// TwinCAT 3 PLC project AstroBROTTests
// Title: AstroBROTTests
// Company: BROT
// ProjectVersion: 0.1.0
// ProgramVersion: 3.1.4024.66
// libraries:
//   AstroBROT, * (BROT)
//   Tc2_Standard, * (Beckhoff Automation GmbH)
//   Tc2_System, * (Beckhoff Automation GmbH)
//   Tc2_Utilities, * (Beckhoff Automation GmbH)
//   Tc3_Module, * (Beckhoff Automation GmbH)
//   TcUnit, * (www.tcunit.org)
// project tree:
//   / PlcTask.TcTTO (not stored)
//   POUs/ FB_DateTime2JD_Tests.TcPOU, FB_ATAN2_Tests.TcPOU, FB_ALTAZ2HADEC_Tests.TcPOU, FB_CO_ABERRATION_Tests.TcPOU, FB_CO_NUTATE_Tests.TcPOU, FB_CO_REFRACT_Tests.TcPOU, FB_DUT1_Tests.TcPOU, FB_Pipeline_Tests.TcPOU, FB_JD2LST_Tests.TcPOU, FB_EQ2HOR_Tests.TcPOU, FB_HOR2EQ_Tests.TcPOU, FB_TEN_Tests.TcPOU, FB_PRECESS_Tests.TcPOU, FB_RADEC2HADEC_Tests.TcPOU, FB_HADEC2RADEC_Tests.TcPOU, FB_SUNPOS_Tests.TcPOU, FB_EdgeCases_Tests.TcPOU, MAIN.TcPOU
// real-time tasks:
//   TASK PlcTask: cycle T#10ms, priority 20, ADS port 350

// ---- POUs/FB_DateTime2JD_Tests.TcPOU
// Tests for AstroBROT.DateTime2JD (TIMESTRUCT, UTC, to Julian Date).
//
// Golden values come from erfa.cal2jd (Gregorian calendar), tolerance 1e-8 days (0.9 ms).
FUNCTION_BLOCK FB_DateTime2JD_Tests EXTENDS TcUnit.FB_TestSuite
VAR
END_VAR

Golden_Dates();
Leap_Years();
Milliseconds();
Out_Of_Range_Fields_Roll_Over();

METHOD PRIVATE Jd : LREAL
VAR_INPUT
	wYear, wMonth, wDay, wHour, wMinute, wSecond, wMilliseconds	: UINT;
END_VAR
VAR
	t	: TIMESTRUCT;
END_VAR
t.wYear := wYear;
t.wMonth := wMonth;
t.wDay := wDay;
t.wHour := wHour;
t.wMinute := wMinute;
t.wSecond := wSecond;
t.wMilliseconds := wMilliseconds;
Jd := AstroBROT.DateTime2JD(epoch := t);
END_METHOD

METHOD PRIVATE CheckNear
VAR_INPUT
	fExpected	: LREAL;
	fActual		: LREAL;
	fDelta		: LREAL;
	sName		: STRING(255);
END_VAR
AssertEquals_LREAL(Expected := fExpected, Actual := fActual, Delta := fDelta, Message := sName);
END_METHOD

METHOD PRIVATE Golden_Dates
VAR
END_VAR
TEST('Golden_Dates');
CheckNear(2451545.0, Jd(2000, 1, 1, 12, 0, 0, 0), 1.0E-8, 'J2000');
CheckNear(2461304.5, Jd(2026, 9, 21, 0, 0, 0, 0), 1.0E-8, '2026-09-21 00:00');
CheckNear(2461305.2710069446, Jd(2026, 9, 21, 18, 30, 15, 0), 1.0E-8, '2026-09-21 18:30:15');
CheckNear(2451544.499988426, Jd(1999, 12, 31, 23, 59, 59, 0), 1.0E-8, '1999-12-31 23:59:59');
CheckNear(2299160.5, Jd(1582, 10, 15, 0, 0, 0, 0), 1.0E-8, '1582-10-15, first Gregorian day');
TEST_FINISHED();
END_METHOD

METHOD PRIVATE Leap_Years
VAR
END_VAR
TEST('Leap_Years');
CheckNear(2460370.0, Jd(2024, 2, 29, 12, 0, 0, 0), 1.0E-8, '2024-02-29 12:00');
CheckNear(1.0, Jd(2024, 3, 1, 0, 0, 0, 0) - Jd(2024, 2, 29, 0, 0, 0, 0), 1.0E-9, '2024 is a leap year');
CheckNear(1.0, Jd(2100, 3, 1, 0, 0, 0, 0) - Jd(2100, 2, 28, 0, 0, 0, 0), 1.0E-9, '2100 is not a leap year');
CheckNear(1.0, Jd(2000, 3, 1, 0, 0, 0, 0) - Jd(2000, 2, 29, 0, 0, 0, 0), 1.0E-9, '2000 is a leap year');
TEST_FINISHED();
END_METHOD

METHOD PRIVATE Milliseconds
VAR
END_VAR
TEST('Milliseconds');
// 500 ms = 5.787037037037037E-6 days
CheckNear(5.787037037037037E-6, Jd(2026, 9, 21, 0, 0, 0, 500) - Jd(2026, 9, 21, 0, 0, 0, 0), 1.0E-9, '500 ms');
CheckNear(1.1574074074074073E-8, Jd(2026, 9, 21, 0, 0, 0, 1) - Jd(2026, 9, 21, 0, 0, 0, 0), 1.0E-9, '1 ms');
TEST_FINISHED();
END_METHOD

METHOD PRIVATE Out_Of_Range_Fields_Roll_Over
VAR
END_VAR
TEST('Out_Of_Range_Fields_Roll_Over');
// documented behaviour, not a feature to rely on
CheckNear(2461406.5, Jd(2026, 13, 1, 0, 0, 0, 0), 1.0E-8, 'month 13 is January of the next year');
CheckNear(2461101.5, Jd(2026, 2, 30, 0, 0, 0, 0), 1.0E-8, '30 February is 2 March');
TEST_FINISHED();
END_METHOD

END_FUNCTION_BLOCK

// ---- POUs/FB_ATAN2_Tests.TcPOU
// Tests for AstroBROT.ATAN2, the four-quadrant arctangent (TwinCAT's PLC has none of its own).
//
// Expected values come from Python math.atan2, tolerance 1e-12 rad. Known difference from IEEE: y = -0.0 with x < 0
// gives +pi (ST cannot tell -0.0 from 0.0), harmless because the callers wrap the angle.
FUNCTION_BLOCK FB_ATAN2_Tests EXTENDS TcUnit.FB_TestSuite
VAR
END_VAR

Quadrants();
Axes();
Origin_Is_Zero();
Close_To_The_Axes();

METHOD PRIVATE CheckAtan2
VAR_INPUT
	fExpected	: LREAL;
	fActual		: LREAL;
	sName		: STRING(255);
END_VAR
AssertEquals_LREAL(Expected := fExpected, Actual := fActual, Delta := 1.0E-12, Message := sName);
END_METHOD

METHOD PRIVATE Quadrants
VAR
END_VAR
TEST('Quadrants');
CheckAtan2(0.7853981633974483, AstroBROT.ATAN2(y := 1.0, x := 1.0), 'q1 (1, 1)');
CheckAtan2(2.5535900500422257, AstroBROT.ATAN2(y := 2.0, x := -3.0), 'q2 (2, -3)');
CheckAtan2(-2.5535900500422257, AstroBROT.ATAN2(y := -2.0, x := -3.0), 'q3 (-2, -3)');
CheckAtan2(-0.5880026035475675, AstroBROT.ATAN2(y := -2.0, x := 3.0), 'q4 (-2, 3)');
CheckAtan2(0.5880026035475675, AstroBROT.ATAN2(y := 2.0, x := 3.0), 'q1 (2, 3)');
CheckAtan2(2.356194490192345, AstroBROT.ATAN2(y := 1.0, x := -1.0), 'q2 (1, -1)');
CheckAtan2(-2.356194490192345, AstroBROT.ATAN2(y := -1.0, x := -1.0), 'q3 (-1, -1)');
CheckAtan2(-0.7853981633974483, AstroBROT.ATAN2(y := -1.0, x := 1.0), 'q4 (-1, 1)');
TEST_FINISHED();
END_METHOD

METHOD PRIVATE Axes
VAR
END_VAR
TEST('Axes');
CheckAtan2(0.0, AstroBROT.ATAN2(y := 0.0, x := 1.0), '+x axis');
CheckAtan2(1.5707963267948966, AstroBROT.ATAN2(y := 1.0, x := 0.0), '+y axis');
CheckAtan2(-1.5707963267948966, AstroBROT.ATAN2(y := -1.0, x := 0.0), '-y axis');
CheckAtan2(3.141592653589793, AstroBROT.ATAN2(y := 0.0, x := -1.0), '-x axis, y = 0 gives +pi');
TEST_FINISHED();
END_METHOD

METHOD PRIVATE Origin_Is_Zero
VAR
END_VAR
TEST('Origin_Is_Zero');
CheckAtan2(0.0, AstroBROT.ATAN2(y := 0.0, x := 0.0), 'origin');
TEST_FINISHED();
END_METHOD

METHOD PRIVATE Close_To_The_Axes
VAR
END_VAR
TEST('Close_To_The_Axes');
CheckAtan2(1.5707963267938967, AstroBROT.ATAN2(y := 1.0, x := 1.0E-12), 'just right of the +y axis');
CheckAtan2(3.141592653588793, AstroBROT.ATAN2(y := 1.0E-12, x := -1.0), 'just above the -x axis');
CheckAtan2(-3.141592653588793, AstroBROT.ATAN2(y := -1.0E-12, x := -1.0), 'just below the -x axis');
TEST_FINISHED();
END_METHOD

END_FUNCTION_BLOCK

// ---- POUs/FB_ALTAZ2HADEC_Tests.TcPOU
// Tests for AstroBROT.FB_ALTAZ2HADEC.
//
// At the celestial pole (az = 0, alt = lat; or az = 180, alt = -lat for the south pole) the argument of ASIN is
// exactly 1 in theory, but rounding gives 1 + 2.2E-16 for many latitudes, and ASIN of that is NaN (issue #18).
FUNCTION_BLOCK FB_ALTAZ2HADEC_Tests EXTENDS TcUnit.FB_TestSuite
VAR
END_VAR

Ordinary_Position();
Pointing_At_The_North_Pole();
Pointing_At_The_South_Pole();

METHOD PRIVATE Ordinary_Position
VAR
	fb	: AstroBROT.FB_ALTAZ2HADEC;
END_VAR
TEST('Ordinary_Position');
// sin(dec) = sin(45)^2 + 0 = 0.5, so dec = 30 deg
fb(alt := 45.0, az := 90.0, lat := 45.0);
AssertEquals_LREAL(Expected := 30.0, Actual := fb.dec, Delta := 1.0E-9, Message := 'dec at alt 45, az 90, lat 45');
TEST_FINISHED();
END_METHOD

METHOD PRIVATE Pointing_At_The_North_Pole
VAR
	fb	: AstroBROT.FB_ALTAZ2HADEC;
END_VAR
TEST('Pointing_At_The_North_Pole');
fb(alt := 45.0, az := 0.0, lat := 45.0);
AssertTrue(Condition := ABS(fb.dec - 90.0) < 1.0E-6, Message := 'lat 45 north pole, dec is 90 (and not NaN)');
fb(alt := 34.0, az := 0.0, lat := 34.0);
AssertTrue(Condition := ABS(fb.dec - 90.0) < 1.0E-6, Message := 'lat 34 north pole, dec is 90 (and not NaN)');
fb(alt := 58.0, az := 0.0, lat := 58.0);
AssertTrue(Condition := ABS(fb.dec - 90.0) < 1.0E-6, Message := 'lat 58 north pole, dec is 90 (and not NaN)');
fb(alt := -34.0, az := 0.0, lat := -34.0);
AssertTrue(Condition := ABS(fb.dec - 90.0) < 1.0E-6, Message := 'lat -34 north pole, dec is 90 (and not NaN)');
TEST_FINISHED();
END_METHOD

METHOD PRIVATE Pointing_At_The_South_Pole
VAR
	fb	: AstroBROT.FB_ALTAZ2HADEC;
END_VAR
TEST('Pointing_At_The_South_Pole');
fb(alt := -45.0, az := 180.0, lat := 45.0);
AssertTrue(Condition := ABS(fb.dec + 90.0) < 1.0E-6, Message := 'lat 45 south pole, dec is -90 (and not NaN)');
fb(alt := -34.0, az := 180.0, lat := 34.0);
AssertTrue(Condition := ABS(fb.dec + 90.0) < 1.0E-6, Message := 'lat 34 south pole, dec is -90 (and not NaN)');
fb(alt := -58.0, az := 180.0, lat := 58.0);
AssertTrue(Condition := ABS(fb.dec + 90.0) < 1.0E-6, Message := 'lat 58 south pole, dec is -90 (and not NaN)');
fb(alt := 34.0, az := 180.0, lat := -34.0);
AssertTrue(Condition := ABS(fb.dec + 90.0) < 1.0E-6, Message := 'lat -34 south pole, dec is -90 (and not NaN)');
TEST_FINISHED();
END_METHOD

END_FUNCTION_BLOCK

// ---- POUs/FB_CO_ABERRATION_Tests.TcPOU
// Tests for AstroBROT.FB_CO_ABERRATION (annual aberration, Meeus chapter 23).
//
// ra/dec are the coordinates precessed to the date, eps = 0 means "calculate the obliquity from jd". Golden values
// come from AstroBROT/testing/golden_astro.py. Tolerance 1e-9 deg (3.6 uas).
FUNCTION_BLOCK FB_CO_ABERRATION_Tests EXTENDS TcUnit.FB_TestSuite
VAR
END_VAR

Golden_Tenerife_2026();
Golden_South_2010();
Eps_Input_Is_Not_Modified();

METHOD PRIVATE CheckNear
VAR_INPUT
	fExpected	: LREAL;
	fActual		: LREAL;
	fDelta		: LREAL;
	sName		: STRING(255);
END_VAR
AssertEquals_LREAL(Expected := fExpected, Actual := fActual, Delta := fDelta, Message := sName);
END_METHOD

METHOD PRIVATE CheckAngle
VAR_INPUT
	fExpected	: LREAL;
	fActual		: LREAL;
	fDelta		: LREAL;
	sName		: STRING(255);
END_VAR
VAR
	fDiff	: LREAL;
END_VAR
// angles in degrees, compared modulo 360 so that 359.9999999 and -1.0E-7 are equal
fDiff := fActual - fExpected;
WHILE fDiff > 180.0 DO fDiff := fDiff - 360.0; END_WHILE
WHILE fDiff < -180.0 DO fDiff := fDiff + 360.0; END_WHILE
AssertEquals_LREAL(Expected := 0.0, Actual := fDiff, Delta := fDelta, Message := sName);
END_METHOD

METHOD PRIVATE Golden_Tenerife_2026
VAR
	fbCalc	: AstroBROT.FB_CO_ABERRATION;
	fbGiven	: AstroBROT.FB_CO_ABERRATION;
END_VAR
TEST('Golden_Tenerife_2026');
fbCalc(jd := 2461300.75, ra := 84.03200262159413, dec := 22.025976570150018, eps := 0.0);
CheckAngle(8.195455011719691e-05, fbCalc.d_ra, 1.0E-9, 'Tenerife_2026 d_ra, eps calculated');
CheckNear(0.00013148215303962214, fbCalc.d_dec, 1.0E-9, 'Tenerife_2026 d_dec, eps calculated');
fbGiven(jd := 2461300.75, ra := 84.03200262159413, dec := 22.025976570150018, eps := 0.40907226011280384);
CheckAngle(8.195455011719691e-05, fbGiven.d_ra, 1.0E-9, 'Tenerife_2026 d_ra, eps given');
CheckNear(0.00013148215303962214, fbGiven.d_dec, 1.0E-9, 'Tenerife_2026 d_dec, eps given');
TEST_FINISHED();
END_METHOD

METHOD PRIVATE Golden_South_2010
VAR
	fbCalc	: AstroBROT.FB_CO_ABERRATION;
	fbGiven	: AstroBROT.FB_CO_ABERRATION;
END_VAR
TEST('Golden_South_2010');
fbCalc(jd := 2455197.5, ra := 312.6725080638107, dec := -47.262327080321406, eps := 0.0);
CheckAngle(-0.007132163801626435, fbCalc.d_ra, 1.0E-9, 'South_2010 d_ra, eps calculated');
CheckNear(-0.0025955563049355266, fbCalc.d_dec, 1.0E-9, 'South_2010 d_dec, eps calculated');
fbGiven(jd := 2455197.5, ra := 312.6725080638107, dec := -47.262327080321406, eps := 0.4090837545317484);
CheckAngle(-0.007132163801626435, fbGiven.d_ra, 1.0E-9, 'South_2010 d_ra, eps given');
CheckNear(-0.0025955563049355266, fbGiven.d_dec, 1.0E-9, 'South_2010 d_dec, eps given');
TEST_FINISHED();
END_METHOD

METHOD PRIVATE Eps_Input_Is_Not_Modified
VAR
	fb	: AstroBROT.FB_CO_ABERRATION;
END_VAR
TEST('Eps_Input_Is_Not_Modified');
// with eps = 0 the block calculates the obliquity itself; it used to store the result in its input, so the
// value of the first jd was reused for every later call
fb(jd := 2461300.75, ra := 84.03200262159413, dec := 22.025976570150018, eps := 0.0);
CheckNear(0.0, fb.eps, 1.0E-15, 'eps stays 0 after the call');
fb(jd := 2455197.5, ra := 312.6725080638107, dec := -47.262327080321406, eps := 0.0);
CheckNear(0.0, fb.eps, 1.0E-15, 'eps stays 0 after the second call');
CheckAngle(-0.007132163801626435, fb.d_ra, 1.0E-9, 'second epoch d_ra');
CheckNear(-0.0025955563049355266, fb.d_dec, 1.0E-9, 'second epoch d_dec');
TEST_FINISHED();
END_METHOD

END_FUNCTION_BLOCK

// ---- POUs/FB_CO_NUTATE_Tests.TcPOU
// Tests for AstroBROT.FB_CO_NUTATE (RA/Dec corrections due to nutation).
//
// Golden values come from AstroBROT/testing/astrobrot_port.py (co_nutate), tolerance 1e-7 deg.
// Issue #10: d_ra was ra2 - ra with ra2 in [0, 360) and ra unwrapped, so ra = -5 gave d_ra = 360.0004 instead of
// 0.00035. The fix wraps d_ra to [-180, 180).
FUNCTION_BLOCK FB_CO_NUTATE_Tests EXTENDS TcUnit.FB_TestSuite
VAR
END_VAR

Golden_Ra_Minus_5();
Golden_Ra_355();
Golden_Ra_0_001();
Golden_Ra_359_999();
Golden_Ra_365();
Golden_South_Ra_Minus_0_001();
Golden_South_Ra_180();
Unwrapped_Ra_Equals_Wrapped_Ra();
D_Ra_Stays_Small_For_Any_Ra();

METHOD PRIVATE CheckNear
VAR_INPUT
	fExpected	: LREAL;
	fActual		: LREAL;
	fDelta		: LREAL;
	sName		: STRING(255);
END_VAR
AssertEquals_LREAL(Expected := fExpected, Actual := fActual, Delta := fDelta, Message := sName);
END_METHOD

METHOD PRIVATE Golden_Ra_Minus_5
VAR
	fb	: AstroBROT.FB_CO_NUTATE;
END_VAR
TEST('Golden_Ra_Minus_5');
fb(jd := 2461000.3, ra := -5.0, dec := 10.0);
CheckNear(0.00035336584255674097, fb.d_ra, 1.0E-7, 'Golden_Ra_Minus_5 d_ra');
CheckNear(0.00012832548964958335, fb.d_dec, 1.0E-7, 'Golden_Ra_Minus_5 d_dec');
TEST_FINISHED();
END_METHOD

METHOD PRIVATE Golden_Ra_355
VAR
	fb	: AstroBROT.FB_CO_NUTATE;
END_VAR
TEST('Golden_Ra_355');
fb(jd := 2461000.3, ra := 355.0, dec := 10.0);
CheckNear(0.0003533658426135844, fb.d_ra, 1.0E-7, 'Golden_Ra_355 d_ra');
CheckNear(0.00012832548964958335, fb.d_dec, 1.0E-7, 'Golden_Ra_355 d_dec');
TEST_FINISHED();
END_METHOD

METHOD PRIVATE Golden_Ra_0_001
VAR
	fb	: AstroBROT.FB_CO_NUTATE;
END_VAR
TEST('Golden_Ra_0_001');
fb(jd := 2461000.3, ra := 0.001, dec := 10.0);
CheckNear(0.00035692751089300145, fb.d_ra, 1.0E-7, 'Golden_Ra_0_001 d_ra');
CheckNear(0.00033419026003578267, fb.d_dec, 1.0E-7, 'Golden_Ra_0_001 d_dec');
TEST_FINISHED();
END_METHOD

METHOD PRIVATE Golden_Ra_359_999
VAR
	fb	: AstroBROT.FB_CO_NUTATE;
END_VAR
TEST('Golden_Ra_359_999');
fb(jd := 2461000.3, ra := 359.999, dec := 10.0);
CheckNear(0.0003569254541275768, fb.d_ra, 1.0E-7, 'Golden_Ra_359_999 d_ra');
CheckNear(0.00033410833518665584, fb.d_dec, 1.0E-7, 'Golden_Ra_359_999 d_dec');
TEST_FINISHED();
END_METHOD

METHOD PRIVATE Golden_Ra_365
VAR
	fb	: AstroBROT.FB_CO_NUTATE;
END_VAR
TEST('Golden_Ra_365');
fb(jd := 2461000.3, ra := 365.0, dec := 10.0);
CheckNear(0.000363636662314093, fb.d_ra, 1.0E-7, 'Golden_Ra_365 d_ra');
CheckNear(0.000537430022859553, fb.d_dec, 1.0E-7, 'Golden_Ra_365 d_dec');
TEST_FINISHED();
END_METHOD

METHOD PRIVATE Golden_South_Ra_Minus_0_001
VAR
	fb	: AstroBROT.FB_CO_NUTATE;
END_VAR
TEST('Golden_South_Ra_Minus_0_001');
fb(jd := 2461000.3, ra := -0.001, dec := -40.0);
CheckNear(0.002740097572001332, fb.d_ra, 1.0E-7, 'Golden_South_Ra_Minus_0_001 d_ra');
CheckNear(0.00033414078795601654, fb.d_dec, 1.0E-7, 'Golden_South_Ra_Minus_0_001 d_dec');
TEST_FINISHED();
END_METHOD

METHOD PRIVATE Golden_South_Ra_180
VAR
	fb	: AstroBROT.FB_CO_NUTATE;
END_VAR
TEST('Golden_South_Ra_180');
fb(jd := 2461000.3, ra := 180.0, dec := -40.0);
CheckNear(-0.001198590003980371, fb.d_ra, 1.0E-7, 'Golden_South_Ra_180 d_ra');
CheckNear(-0.00033414331457493063, fb.d_dec, 1.0E-7, 'Golden_South_Ra_180 d_dec');
TEST_FINISHED();
END_METHOD

METHOD PRIVATE Unwrapped_Ra_Equals_Wrapped_Ra
VAR
	fbA, fbB	: AstroBROT.FB_CO_NUTATE;
END_VAR
TEST('Unwrapped_Ra_Equals_Wrapped_Ra');
// ra and ra + 360 are the same direction, so the RA correction must agree (before the fix ra = -5 gave 360.0004)
fbA(jd := 2461000.3, ra := -5.0, dec := 10.0);
fbB(jd := 2461000.3, ra := 355.0, dec := 10.0);
CheckNear(fbB.d_ra, fbA.d_ra, 1.0E-9, 'd_ra(-5) = d_ra(355)');
CheckNear(fbB.d_dec, fbA.d_dec, 1.0E-9, 'd_dec(-5) = d_dec(355)');
TEST_FINISHED();
END_METHOD

METHOD PRIVATE D_Ra_Stays_Small_For_Any_Ra
VAR
	fb	: AstroBROT.FB_CO_NUTATE;
	i	: INT;
	fMax, fAbs	: LREAL;
END_VAR
TEST('D_Ra_Stays_Small_For_Any_Ra');
// FB_HADEC2RADEC can pass any ra in (-360, 360); nutation moves RA by at most ~0.011 deg at |dec| <= 60
fMax := 0.0;
FOR i := -24 TO 48 DO
	fb(jd := 2461000.3, ra := INT_TO_LREAL(i) * 15.0 + 0.5, dec := 10.0);
	fAbs := ABS(fb.d_ra);
	IF fAbs > fMax THEN fMax := fAbs; END_IF
END_FOR
AssertTrue(Condition := fMax < 0.02, Message := 'max |d_ra| over ra -360..720 is below 0.02 deg');
TEST_FINISHED();
END_METHOD

END_FUNCTION_BLOCK

// ---- POUs/FB_CO_REFRACT_Tests.TcPOU
// Tests for AstroBROT.FB_CO_REFRACT and CO_REFRACT_FORWARD (atmospheric refraction).
//
//   to_observed = FALSE: old_alt is the observed altitude, new_alt the geometric one (refraction removed)
//   to_observed = TRUE : old_alt is geometric, new_alt observed (iterated)
//
// Golden values come from AstroBROT/testing/golden_astro.py (temperature in degrees Celsius), tolerance 1e-7 deg.
// The refraction model is CO_REFRACT_FORWARD: rational formula below 14 deg, eraRefco (dry) from 16 deg, blend between (#11).
FUNCTION_BLOCK FB_CO_REFRACT_Tests EXTENDS TcUnit.FB_TestSuite
VAR
END_VAR

Golden_Observed_To_Geometric();
Golden_Geometric_To_Observed();
Temperature_Zero_Celsius_Is_Used();
No_State_Is_Kept_Between_Calls();
Out_Of_Range_Altitude_Passes_Through();
Zero_Or_Negative_Epsilon_Terminates();
Forward_Values();
Continuous_And_Decreasing();
Clamped_Flag();

METHOD PRIVATE CheckNear
VAR_INPUT
	fExpected	: LREAL;
	fActual		: LREAL;
	fDelta		: LREAL;
	sName		: STRING(255);
END_VAR
AssertEquals_LREAL(Expected := fExpected, Actual := fActual, Delta := fDelta, Message := sName);
END_METHOD

METHOD PRIVATE CheckAngle
VAR_INPUT
	fExpected	: LREAL;
	fActual		: LREAL;
	fDelta		: LREAL;
	sName		: STRING(255);
END_VAR
VAR
	fDiff	: LREAL;
END_VAR
// angles in degrees, compared modulo 360 so that 359.9999999 and -1.0E-7 are equal
fDiff := fActual - fExpected;
WHILE fDiff > 180.0 DO fDiff := fDiff - 360.0; END_WHILE
WHILE fDiff < -180.0 DO fDiff := fDiff + 360.0; END_WHILE
AssertEquals_LREAL(Expected := 0.0, Actual := fDiff, Delta := fDelta, Message := sName);
END_METHOD

METHOD PRIVATE Golden_Observed_To_Geometric
VAR
	fb	: AstroBROT.FB_CO_REFRACT;
END_VAR
TEST('Golden_Observed_To_Geometric');
fb(old_alt := 45.0, altitude := 0.0, pressure := 0.0, to_observed := FALSE);
CheckNear(44.98388737240353, fb.new_alt, 1.0E-7, 'alt45_sea to geometric');
fb(old_alt := 10.0, altitude := 0.0, pressure := 0.0, to_observed := FALSE);
CheckNear(9.912032655050567, fb.new_alt, 1.0E-7, 'alt10_sea to geometric');
fb(old_alt := 3.0, altitude := 2400.0, pressure := 0.0, to_observed := FALSE);
CheckNear(2.8120678712676828, fb.new_alt, 1.0E-7, 'alt3_high to geometric');
fb(old_alt := 20.0, altitude := 0.0, pressure := 1000.0, temperature := 0.0, temperature_set := TRUE, to_observed := FALSE);
CheckNear(19.954879536938076, fb.new_alt, 1.0E-7, 'alt20_P_T0 to geometric');
fb(old_alt := 20.0, altitude := 0.0, pressure := 900.0, temperature := -15.0, temperature_set := TRUE, to_observed := FALSE);
CheckNear(19.957009525944056, fb.new_alt, 1.0E-7, 'alt20_P_Tminus15 to geometric');
TEST_FINISHED();
END_METHOD

METHOD PRIVATE Golden_Geometric_To_Observed
VAR
	fb	: AstroBROT.FB_CO_REFRACT;
END_VAR
TEST('Golden_Geometric_To_Observed');
fb(old_alt := 45.0, altitude := 0.0, pressure := 0.0, to_observed := TRUE, epsilon := 0.001);
CheckNear(45.01610359317409, fb.new_alt, 1.0E-7, 'alt45_sea to observed');
fb(old_alt := 10.0, altitude := 0.0, pressure := 0.0, to_observed := TRUE, epsilon := 0.001);
CheckNear(10.087240824501489, fb.new_alt, 1.0E-7, 'alt10_sea to observed');
fb(old_alt := 3.0, altitude := 2400.0, pressure := 0.0, to_observed := TRUE, epsilon := 0.001);
CheckNear(3.180753517200842, fb.new_alt, 1.0E-7, 'alt3_high to observed');
fb(old_alt := 20.0, altitude := 0.0, pressure := 1000.0, temperature := 0.0, temperature_set := TRUE, to_observed := TRUE, epsilon := 0.001);
CheckNear(20.045012197500732, fb.new_alt, 1.0E-7, 'alt20_P_T0 to observed');
fb(old_alt := 20.0, altitude := 0.0, pressure := 900.0, temperature := -15.0, temperature_set := TRUE, to_observed := TRUE, epsilon := 0.001);
CheckNear(20.042892076742575, fb.new_alt, 1.0E-7, 'alt20_P_Tminus15 to observed');
TEST_FINISHED();
END_METHOD

METHOD PRIVATE Temperature_Zero_Celsius_Is_Used
VAR
	fbT0	: AstroBROT.FB_CO_REFRACT;
	fbEst	: AstroBROT.FB_CO_REFRACT;
END_VAR
TEST('Temperature_Zero_Celsius_Is_Used');
fbT0(old_alt := 20.0, altitude := 0.0, pressure := 1000.0, temperature := 0.0, temperature_set := TRUE, to_observed := FALSE);
fbEst(old_alt := 20.0, altitude := 0.0, pressure := 1000.0, to_observed := FALSE);
CheckNear(19.954879536938076, fbT0.new_alt, 1.0E-7, '0.0 C with temperature_set');
// without temperature_set the temperature is estimated from the altitude (10 C at sea level), which must differ
AssertTrue(Condition := ABS(fbEst.new_alt - fbT0.new_alt) > 1.0E-5, Message := 'estimated temperature differs from 0.0 C');
TEST_FINISHED();
END_METHOD

METHOD PRIVATE No_State_Is_Kept_Between_Calls
VAR
	fb	: AstroBROT.FB_CO_REFRACT;
END_VAR
TEST('No_State_Is_Kept_Between_Calls');
// the estimated pressure and temperature of the first call (sea level) must not leak into the second (2400 m)
fb(old_alt := 45.0, altitude := 0.0, pressure := 0.0, to_observed := FALSE);
fb(old_alt := 3.0, altitude := 2400.0, pressure := 0.0, to_observed := FALSE);
CheckNear(2.8120678712676828, fb.new_alt, 1.0E-7, 'high site after sea level call');
CheckNear(0.0, fb.pressure, 1.0E-15, 'pressure input unchanged');
CheckNear(0.0, fb.temperature, 1.0E-15, 'temperature input unchanged');
TEST_FINISHED();
END_METHOD

METHOD PRIVATE Out_Of_Range_Altitude_Passes_Through
VAR
	fb	: AstroBROT.FB_CO_REFRACT;
END_VAR
TEST('Out_Of_Range_Altitude_Passes_Through');
fb(old_alt := 2.0E6, to_observed := TRUE);
CheckNear(2.0E6, fb.new_alt, 1.0E-15, '2e6 deg to observed');
fb(old_alt := -1.0E9, to_observed := TRUE);
CheckNear(-1.0E9, fb.new_alt, 1.0E-15, '-1e9 deg to observed');
fb(old_alt := 2.0E6, to_observed := FALSE);
CheckNear(2.0E6, fb.new_alt, 1.0E-15, '2e6 deg to geometric');
TEST_FINISHED();
END_METHOD

METHOD PRIVATE Zero_Or_Negative_Epsilon_Terminates
VAR
	fb	: AstroBROT.FB_CO_REFRACT;
END_VAR
TEST('Zero_Or_Negative_Epsilon_Terminates');
// epsilon <= 0 could never satisfy the exit condition of the iteration; it is clamped to 0.001 arcsec
fb(old_alt := 10.0, altitude := 0.0, pressure := 0.0, to_observed := TRUE, epsilon := 0.0);
CheckNear(10.087240824501489, fb.new_alt, 1.0E-7, 'epsilon 0');
fb(old_alt := 10.0, altitude := 0.0, pressure := 0.0, to_observed := TRUE, epsilon := -5.0);
CheckNear(10.087240824501489, fb.new_alt, 1.0E-7, 'epsilon -5');
TEST_FINISHED();
END_METHOD

METHOD PRIVATE Forward_Values
VAR
END_VAR
TEST('Forward_Values');
// refraction in degrees from CO_REFRACT_FORWARD, values from testing/astrobrot_port.py (agrees with erfa.refco from 16 deg up)
CheckNear(0.163267493516567, AstroBROT.CO_REFRACT_FORWARD(a := 5.0, P := 1010.0, T := 10.0), 1.0E-9, 'a5 P1010 T10');
CheckNear(0.08796734494943341, AstroBROT.CO_REFRACT_FORWARD(a := 10.0, P := 1010.0, T := 10.0), 1.0E-9, 'a10 P1010 T10');
CheckNear(0.0634207907895386, AstroBROT.CO_REFRACT_FORWARD(a := 14.0, P := 1010.0, T := 10.0), 1.0E-9, 'a14 P1010 T10');
CheckNear(0.05924934349202771, AstroBROT.CO_REFRACT_FORWARD(a := 15.0, P := 1010.0, T := 10.0), 1.0E-9, 'a15 P1010 T10');
CheckNear(0.055488304257851416, AstroBROT.CO_REFRACT_FORWARD(a := 16.0, P := 1010.0, T := 10.0), 1.0E-9, 'a16 P1010 T10');
CheckNear(0.027845320022875337, AstroBROT.CO_REFRACT_FORWARD(a := 30.0, P := 1010.0, T := 10.0), 1.0E-9, 'a30 P1010 T10');
CheckNear(0.016112627596470155, AstroBROT.CO_REFRACT_FORWARD(a := 45.0, P := 1010.0, T := 10.0), 1.0E-9, 'a45 P1010 T10');
CheckNear(0.009309582059912834, AstroBROT.CO_REFRACT_FORWARD(a := 60.0, P := 1010.0, T := 10.0), 1.0E-9, 'a60 P1010 T10');
CheckNear(0.0028441768234894497, AstroBROT.CO_REFRACT_FORWARD(a := 80.0, P := 1010.0, T := 10.0), 1.0E-9, 'a80 P1010 T10');
CheckNear(0.159583354818749, AstroBROT.CO_REFRACT_FORWARD(a := 5.0, P := 900.0, T := -15.0), 1.0E-9, 'a5 P900 T-15');
CheckNear(0.08598235765838011, AstroBROT.CO_REFRACT_FORWARD(a := 10.0, P := 900.0, T := -15.0), 1.0E-9, 'a10 P900 T-15');
CheckNear(0.06198969765175947, AstroBROT.CO_REFRACT_FORWARD(a := 14.0, P := 900.0, T := -15.0), 1.0E-9, 'a14 P900 T-15');
CheckNear(0.057958476783226534, AstroBROT.CO_REFRACT_FORWARD(a := 15.0, P := 900.0, T := -15.0), 1.0E-9, 'a15 P900 T-15');
CheckNear(0.05431185364376681, AstroBROT.CO_REFRACT_FORWARD(a := 16.0, P := 900.0, T := -15.0), 1.0E-9, 'a16 P900 T-15');
CheckNear(0.02722749052714757, AstroBROT.CO_REFRACT_FORWARD(a := 30.0, P := 900.0, T := -15.0), 1.0E-9, 'a30 P900 T-15');
CheckNear(0.015751696957665602, AstroBROT.CO_REFRACT_FORWARD(a := 45.0, P := 900.0, T := -15.0), 1.0E-9, 'a45 P900 T-15');
CheckNear(0.009100385246363576, AstroBROT.CO_REFRACT_FORWARD(a := 60.0, P := 900.0, T := -15.0), 1.0E-9, 'a60 P900 T-15');
CheckNear(0.0027801739663453123, AstroBROT.CO_REFRACT_FORWARD(a := 80.0, P := 900.0, T := -15.0), 1.0E-9, 'a80 P900 T-15');
TEST_FINISHED();
END_METHOD

METHOD PRIVATE Continuous_And_Decreasing
VAR
	k, i	: INT;
	P, T, prev, cur	: LREAL;
	bOk, bDown	: BOOL;
END_VAR
TEST('Continuous_And_Decreasing');
// the branches are blended between 14 and 16 deg, there must be no step (it was 5.2 arcsec at 15 deg, issue #11)
bOk := TRUE; bDown := TRUE;
FOR k := 0 TO 1 DO
	IF k = 0 THEN
		P := 1010.0; T := 10.0;
	ELSE
		P := 900.0; T := -15.0;
	END_IF
	prev := AstroBROT.CO_REFRACT_FORWARD(a := 10.0, P := P, T := T);
	FOR i := 1 TO 1580 DO
		cur := AstroBROT.CO_REFRACT_FORWARD(a := 10.0 + INT_TO_LREAL(i) * 0.05, P := P, T := T);
		IF NOT (ABS(prev - cur) < 6.0E-4) THEN bOk := FALSE; END_IF
		IF NOT (cur < prev) THEN bDown := FALSE; END_IF
		prev := cur;
	END_FOR
END_FOR
AssertTrue(Condition := bOk, Message := 'no step larger than 6E-4 deg per 0.05 deg between 10 and 89 deg');
AssertTrue(Condition := bDown, Message := 'refraction decreases with altitude');
TEST_FINISHED();
END_METHOD

METHOD PRIVATE Clamped_Flag
VAR
	fb	: AstroBROT.FB_CO_REFRACT;
END_VAR
TEST('Clamped_Flag');
fb(old_alt := 45.0, altitude := 0.0, pressure := 0.0, to_observed := FALSE);
AssertFalse(Condition := fb.clamped, Message := 'ordinary input is not clamped');
fb(old_alt := 45.0, altitude := 0.0, pressure := 0.0, to_observed := TRUE);
AssertFalse(Condition := fb.clamped, Message := 'ordinary input is not clamped, to observed');
fb(old_alt := -1.0, altitude := 0.0, pressure := 0.0, to_observed := FALSE);
AssertTrue(Condition := fb.clamped, Message := 'below the horizon');
fb(old_alt := 45.0, altitude := 0.0, pressure := 500.0, to_observed := FALSE);
AssertTrue(Condition := fb.clamped, Message := 'pressure below 600 mbar');
fb(old_alt := 45.0, altitude := 0.0, pressure := 1000.0, temperature := 50.0, temperature_set := TRUE, to_observed := FALSE);
AssertTrue(Condition := fb.clamped, Message := 'temperature above 40 degC');
fb(old_alt := 2.0E6, to_observed := TRUE);
AssertTrue(Condition := fb.clamped, Message := 'rejected altitude, passed through unchanged');
TEST_FINISHED();
END_METHOD

END_FUNCTION_BLOCK

// ---- POUs/FB_DUT1_Tests.TcPOU
// Tests for the dut1 input (UT1-UTC in seconds, issue #12) of FB_RADEC2HADEC and FB_HADEC2RADEC.
//
// The golden tests for FB_EQ2HOR and FB_HOR2EQ live in their own suites. Here the effect is checked relative to
// dut1 = 0: only the sidereal time changes, so the hour angle grows by dut1 * 360.98564736629 / 86400 deg and
// the right ascension shrinks by the same amount.
FUNCTION_BLOCK FB_DUT1_Tests EXTENDS TcUnit.FB_TestSuite
VAR
END_VAR

RADEC2HADEC_Hour_Angle_Follows_Dut1();
HADEC2RADEC_Right_Ascension_Follows_Dut1();
Round_Trip_With_Dut1();
Inputs_Are_Not_Modified();

METHOD PRIVATE CheckNear
VAR_INPUT
	fExpected	: LREAL;
	fActual		: LREAL;
	fDelta		: LREAL;
	sName		: STRING(255);
END_VAR
AssertEquals_LREAL(Expected := fExpected, Actual := fActual, Delta := fDelta, Message := sName);
END_METHOD

METHOD PRIVATE CheckAngle
VAR_INPUT
	fExpected	: LREAL;
	fActual		: LREAL;
	fDelta		: LREAL;
	sName		: STRING(255);
END_VAR
VAR
	fDiff	: LREAL;
END_VAR
// angles in degrees, compared modulo 360 so that 359.9999999 and -1.0E-7 are equal
fDiff := fActual - fExpected;
WHILE fDiff > 180.0 DO fDiff := fDiff - 360.0; END_WHILE
WHILE fDiff < -180.0 DO fDiff := fDiff + 360.0; END_WHILE
AssertEquals_LREAL(Expected := 0.0, Actual := fDiff, Delta := fDelta, Message := sName);
END_METHOD

METHOD PRIVATE RADEC2HADEC_Hour_Angle_Follows_Dut1
VAR
	fb0	: AstroBROT.FB_RADEC2HADEC;
	fbP	: AstroBROT.FB_RADEC2HADEC;
	fbM	: AstroBROT.FB_RADEC2HADEC;
	fDelta	: LREAL;
END_VAR
TEST('RADEC2HADEC_Hour_Angle_Follows_Dut1');
// jd + dut1 / 86400 is quantised to about 40 us (up to 1.7E-7 deg), so the tolerance is 5E-7 deg
fDelta := 0.9 * 360.98564736629 / 86400.0;
fb0(jd := 2461300.75, ra := 83.63, dec := 22.01, lon := -16.5, dut1 := 0.0);
fbP(jd := 2461300.75, ra := 83.63, dec := 22.01, lon := -16.5, dut1 := 0.9);
fbM(jd := 2461300.75, ra := 83.63, dec := 22.01, lon := -16.5, dut1 := -0.9);
CheckAngle(fb0.ha_out + fDelta, fbP.ha_out, 5.0E-7, 'ha +0.9 s');
CheckAngle(fb0.ha_out - fDelta, fbM.ha_out, 5.0E-7, 'ha -0.9 s');
CheckNear(fb0.dec_out, fbP.dec_out, 1.0E-9, 'dec is independent of dut1');
TEST_FINISHED();
END_METHOD

METHOD PRIVATE HADEC2RADEC_Right_Ascension_Follows_Dut1
VAR
	fb0	: AstroBROT.FB_HADEC2RADEC;
	fbP	: AstroBROT.FB_HADEC2RADEC;
	fbM	: AstroBROT.FB_HADEC2RADEC;
	fDelta	: LREAL;
END_VAR
TEST('HADEC2RADEC_Right_Ascension_Follows_Dut1');
// nutation and aberration depend slightly on RA, so the tolerance is 1e-6 deg, far below the 3.8e-3 deg shift
fDelta := 0.9 * 360.98564736629 / 86400.0;
fb0(jd := 2461300.75, ha := 345.0, dec := 22.01, lon := -16.5, dut1 := 0.0);
fbP(jd := 2461300.75, ha := 345.0, dec := 22.01, lon := -16.5, dut1 := 0.9);
fbM(jd := 2461300.75, ha := 345.0, dec := 22.01, lon := -16.5, dut1 := -0.9);
CheckAngle(fb0.ra_out + fDelta, fbP.ra_out, 1.0E-6, 'ra +0.9 s');
CheckAngle(fb0.ra_out - fDelta, fbM.ra_out, 1.0E-6, 'ra -0.9 s');
TEST_FINISHED();
END_METHOD

METHOD PRIVATE Round_Trip_With_Dut1
VAR
	fbFwd	: AstroBROT.FB_RADEC2HADEC;
	fbBack	: AstroBROT.FB_HADEC2RADEC;
END_VAR
TEST('Round_Trip_With_Dut1');
// the same dut1 in both directions cancels
fbFwd(jd := 2461300.75, ra := 83.63, dec := 22.01, lon := -16.5, dut1 := 0.7);
fbBack(jd := 2461300.75, ha := fbFwd.ha_out, dec := fbFwd.dec_out, lon := -16.5, dut1 := 0.7);
CheckAngle(83.63, fbBack.ra_out, 1.0E-6, 'ra');
CheckNear(22.01, fbBack.dec_out, 1.0E-6, 'dec');
TEST_FINISHED();
END_METHOD

METHOD PRIVATE Inputs_Are_Not_Modified
VAR
	fbFwd	: AstroBROT.FB_RADEC2HADEC;
	fbBack	: AstroBROT.FB_HADEC2RADEC;
END_VAR
TEST('Inputs_Are_Not_Modified');
fbFwd(jd := 2461300.75, ra := 83.63, dec := 22.01, lon := -16.5, dut1 := 0.7);
CheckNear(0.7, fbFwd.dut1, 0.0, 'FB_RADEC2HADEC dut1');
fbBack(jd := 2461300.75, ha := 345.0, dec := 22.01, lon := -16.5, dut1 := 0.7);
CheckNear(0.7, fbBack.dut1, 0.0, 'FB_HADEC2RADEC dut1');
TEST_FINISHED();
END_METHOD

END_FUNCTION_BLOCK

// ---- POUs/FB_Pipeline_Tests.TcPOU
// Tests for the shared building blocks of the apparent-place pipeline (issue #14, finding M7): the helper functions
// JD2OBLIQUITY, JD2JEPOCH and LMST2LAST, the precess / nutate / aberration switches of FB_RADEC2HADEC and
// FB_HADEC2RADEC, the nut_given input of FB_CO_NUTATE, and that FB_EQ2HOR and FB_HOR2EQ are exactly the composition of
// these blocks with FB_HADEC2ALTAZ / FB_ALTAZ2HADEC.
//
// The golden numbers of the helpers come from the formulas themselves (Python) and are cross-checked against
// erfa.obl06 (the polynomial differs from IAU 2006 by 0.05 arcsec). The switch tests are relative: with everything
// off the blocks only apply the sidereal time, and each switch on its own adds exactly the correction that the
// separate FB_PRECESS / FB_CO_NUTATE / FB_CO_ABERRATION returns.
FUNCTION_BLOCK FB_Pipeline_Tests EXTENDS TcUnit.FB_TestSuite
VAR
END_VAR

JD2OBLIQUITY_Golden();
JD2JEPOCH_Golden();
LMST2LAST_Golden();
CO_NUTATE_Given_Nutation_Is_Used_Not_Evaluated();
RADEC2HADEC_All_Switches_Off_Only_Applies_Sidereal_Time();
RADEC2HADEC_Each_Switch_Applies_Exactly_One_Correction();
RADEC2HADEC_Switching_Off_Does_Not_Keep_The_Last_Correction();
RADEC2HADEC_Cyclic_Calls_With_Inputs_Set_Once_Are_Stable();
HADEC2RADEC_All_Switches_Off_Only_Applies_Sidereal_Time();
HADEC2RADEC_Each_Switch_Applies_Exactly_One_Correction();
HADEC2RADEC_Right_Ascension_Is_Wrapped_Without_Precession();
HADEC2RADEC_Switching_Off_Does_Not_Keep_The_Last_Correction();
EQ2HOR_Is_The_Composition_Of_Its_Parts();
HOR2EQ_Is_The_Composition_Of_Its_Parts();

METHOD PRIVATE CheckNear
VAR_INPUT
	fExpected	: LREAL;
	fActual		: LREAL;
	fDelta		: LREAL;
	sName		: STRING(255);
END_VAR
AssertEquals_LREAL(Expected := fExpected, Actual := fActual, Delta := fDelta, Message := sName);
END_METHOD

METHOD PRIVATE CheckAngle
VAR_INPUT
	fExpected	: LREAL;
	fActual		: LREAL;
	fDelta		: LREAL;
	sName		: STRING(255);
END_VAR
VAR
	fDiff	: LREAL;
END_VAR
// angles in degrees, compared modulo 360 so that 359.9999999 and -1.0E-7 are equal
fDiff := fActual - fExpected;
WHILE fDiff > 180.0 DO fDiff := fDiff - 360.0; END_WHILE
WHILE fDiff < -180.0 DO fDiff := fDiff + 360.0; END_WHILE
AssertEquals_LREAL(Expected := 0.0, Actual := fDiff, Delta := fDelta, Message := sName);
END_METHOD

METHOD PRIVATE ApparentSidereal : LREAL
VAR_INPUT
	jd		: LREAL;
	lon		: LREAL;
END_VAR
VAR
	nut		: AstroBROT.FB_IAU2000B;
END_VAR
// local apparent sidereal time in degrees, built from the pieces the blocks use
nut(jd := jd);
ApparentSidereal := AstroBROT.LMST2LAST(
	lmst := AstroBROT.JD2LST(jd := jd, lon := lon, dut1 := 0.0),
	d_psi := nut.d_psi,
	eps := AstroBROT.JD2OBLIQUITY(jd := jd, d_eps := nut.d_eps));
END_METHOD

METHOD PRIVATE JD2OBLIQUITY_Golden
TEST('JD2OBLIQUITY_Golden');
CheckNear(0.4090928040284035, AstroBROT.JD2OBLIQUITY(jd := 2451545.0, d_eps := 0.0), 1.0E-12, 'J2000, no nutation');
CheckNear(0.40903218198173297, AstroBROT.JD2OBLIQUITY(jd := 2461300.75, d_eps := 0.0), 1.0E-12, '2026-09-21, no nutation');
CheckNear(0.40894733958753876, AstroBROT.JD2OBLIQUITY(jd := 2461300.75, d_eps := -17.5), 1.0E-12, 'd_eps is added in arcsec');
CheckNear(0.40916089319108967, AstroBROT.JD2OBLIQUITY(jd := 2440587.5, d_eps := 0.0), 1.0E-12, '1970');
CheckNear(AstroBROT.JD2OBLIQUITY(jd := 2461300.75, d_eps := 0.0) + PI / 180.0, AstroBROT.JD2OBLIQUITY(jd := 2461300.75, d_eps := 3600.0), 1.0E-12, '3600 arcsec is one degree');
// erfa.obl06 (IAU 2006 mean obliquity): 0.4090926006005829 and 0.4090319505229558, 0.05 arcsec = 2.3E-7 rad away
CheckNear(0.4090926006005829, AstroBROT.JD2OBLIQUITY(jd := 2451545.0, d_eps := 0.0), 5.0E-7, 'erfa J2000');
CheckNear(0.4090319505229558, AstroBROT.JD2OBLIQUITY(jd := 2461300.75, d_eps := 0.0), 5.0E-7, 'erfa 2026-09-21');
TEST_FINISHED();
END_METHOD

METHOD PRIVATE JD2JEPOCH_Golden
TEST('JD2JEPOCH_Golden');
CheckNear(2000.0, AstroBROT.JD2JEPOCH(jd := 2451545.0), 1.0E-9, 'J2000');
CheckNear(2001.0, AstroBROT.JD2JEPOCH(jd := 2451910.25), 1.0E-9, 'one Julian year later');
CheckNear(2026.709787816564, AstroBROT.JD2JEPOCH(jd := 2461300.75), 1.0E-9, '2026-09-21');
CheckNear(1970.0, AstroBROT.JD2JEPOCH(jd := 2440587.5), 1.0E-9, '1970');
TEST_FINISHED();
END_METHOD

METHOD PRIVATE LMST2LAST_Golden
TEST('LMST2LAST_Golden');
CheckNear(100.0, AstroBROT.LMST2LAST(lmst := 100.0, d_psi := 0.0, eps := 0.4), 1.0E-12, 'no nutation');
CheckNear(101.0, AstroBROT.LMST2LAST(lmst := 100.0, d_psi := 3600.0, eps := 0.0), 1.0E-12, 'eps 0: d_psi in full, 3600 arcsec is one degree');
CheckNear(99.5, AstroBROT.LMST2LAST(lmst := 100.0, d_psi := -3600.0, eps := PI / 3.0), 1.0E-12, 'cos(60 deg) = 0.5');
CheckNear(100.0, AstroBROT.LMST2LAST(lmst := 100.0, d_psi := 3600.0, eps := PI / 2.0), 1.0E-12, 'eps 90 deg: no correction');
CheckNear(100.0 + -14.0 * COS(0.409) / 3600.0, AstroBROT.LMST2LAST(lmst := 100.0, d_psi := -14.0, eps := 0.409), 1.0E-12, 'typical values');
TEST_FINISHED();
END_METHOD

METHOD PRIVATE CO_NUTATE_Given_Nutation_Is_Used_Not_Evaluated
VAR
	fbA	: AstroBROT.FB_CO_NUTATE;
	fbB	: AstroBROT.FB_CO_NUTATE;
	fbC	: AstroBROT.FB_CO_NUTATE;
END_VAR
TEST('CO_NUTATE_Given_Nutation_Is_Used_Not_Evaluated');
fbA(jd := 2461300.75, ra := 83.63, dec := 22.01);
AssertTrue(Condition := ABS(fbA.d_ra) > 1.0E-6, Message := 'nutation is evaluated by default');
// the nutation of the same date passed in gives the same corrections
fbB(jd := 2461300.75, ra := 83.63, dec := 22.01, nut_given := TRUE, d_psi_in := fbA.d_psi, d_eps_in := fbA.d_eps);
CheckNear(fbA.d_ra, fbB.d_ra, 1.0E-12, 'd_ra');
CheckNear(fbA.d_dec, fbB.d_dec, 1.0E-12, 'd_dec');
CheckNear(fbA.d_psi, fbB.d_psi, 0.0, 'd_psi');
CheckNear(fbA.d_eps, fbB.d_eps, 0.0, 'd_eps');
CheckNear(fbA.eps, fbB.eps, 1.0E-12, 'eps');
// a given zero nutation is used as it is: nothing is looked up for jd
fbC(jd := 2461300.75, ra := 83.63, dec := 22.01, nut_given := TRUE, d_psi_in := 0.0, d_eps_in := 0.0);
CheckNear(0.0, fbC.d_psi, 0.0, 'given d_psi');
CheckNear(0.0, fbC.d_ra, 1.0E-9, 'no nutation: d_ra');
CheckNear(0.0, fbC.d_dec, 1.0E-9, 'no nutation: d_dec');
CheckNear(AstroBROT.JD2OBLIQUITY(jd := 2461300.75, d_eps := 0.0), fbC.eps, 1.0E-12, 'eps is the mean obliquity');
TEST_FINISHED();
END_METHOD

METHOD PRIVATE RADEC2HADEC_All_Switches_Off_Only_Applies_Sidereal_Time
VAR
	fb		: AstroBROT.FB_RADEC2HADEC;
	fLast	: LREAL;
END_VAR
TEST('RADEC2HADEC_All_Switches_Off_Only_Applies_Sidereal_Time');
fLast := ApparentSidereal(2461300.75, -16.5);
fb(jd := 2461300.75, ra := 83.63, dec := 22.01, lon := -16.5, precess := FALSE, nutate := FALSE, aberration := FALSE);
CheckAngle(fLast - 83.63, fb.ha_out, 1.0E-9, 'ha = LAST - ra');
CheckNear(22.01, fb.dec_out, 0.0, 'dec unchanged');
TEST_FINISHED();
END_METHOD

METHOD PRIVATE RADEC2HADEC_Each_Switch_Applies_Exactly_One_Correction
VAR
	fbOff		: AstroBROT.FB_RADEC2HADEC;
	fbPre		: AstroBROT.FB_RADEC2HADEC;
	fbNut		: AstroBROT.FB_RADEC2HADEC;
	fbAbr		: AstroBROT.FB_RADEC2HADEC;
	fbPrecess	: AstroBROT.FB_PRECESS;
	nut			: AstroBROT.FB_CO_NUTATE;
	abr			: AstroBROT.FB_CO_ABERRATION;
END_VAR
TEST('RADEC2HADEC_Each_Switch_Applies_Exactly_One_Correction');
fbOff(jd := 2461300.75, ra := 83.63, dec := 22.01, lon := -16.5, precess := FALSE, nutate := FALSE, aberration := FALSE);
fbPre(jd := 2461300.75, ra := 83.63, dec := 22.01, lon := -16.5, precess := TRUE, nutate := FALSE, aberration := FALSE);
fbNut(jd := 2461300.75, ra := 83.63, dec := 22.01, lon := -16.5, precess := FALSE, nutate := TRUE, aberration := FALSE);
fbAbr(jd := 2461300.75, ra := 83.63, dec := 22.01, lon := -16.5, precess := FALSE, nutate := FALSE, aberration := TRUE);
fbPrecess(ra := 83.63, dec := 22.01, equinox1 := 2000.0, equinox2 := AstroBROT.JD2JEPOCH(jd := 2461300.75));
nut(jd := 2461300.75, ra := 83.63, dec := 22.01);
abr(jd := 2461300.75, ra := 83.63, dec := 22.01);
// the corrections must be big enough for the comparisons below to mean something
AssertTrue(Condition := ABS(fbPrecess.ra_precessed - 83.63) > 1.0E-3, Message := 'precession is not negligible');
AssertTrue(Condition := ABS(nut.d_ra) > 1.0E-5, Message := 'nutation is not negligible');
AssertTrue(Condition := ABS(abr.d_ra) > 1.0E-5, Message := 'aberration is not negligible');
// ha = LAST - ra_apparent, so a correction d_ra to ra lowers ha by d_ra
CheckAngle(fbOff.ha_out - (fbPrecess.ra_precessed - 83.63), fbPre.ha_out, 1.0E-9, 'precession only: ha');
CheckNear(fbPrecess.dec_precessed, fbPre.dec_out, 1.0E-9, 'precession only: dec');
CheckAngle(fbOff.ha_out - nut.d_ra, fbNut.ha_out, 1.0E-9, 'nutation only: ha');
CheckNear(22.01 + nut.d_dec, fbNut.dec_out, 1.0E-9, 'nutation only: dec');
CheckAngle(fbOff.ha_out - abr.d_ra, fbAbr.ha_out, 1.0E-9, 'aberration only: ha');
CheckNear(22.01 + abr.d_dec, fbAbr.dec_out, 1.0E-9, 'aberration only: dec');
TEST_FINISHED();
END_METHOD

METHOD PRIVATE RADEC2HADEC_Switching_Off_Does_Not_Keep_The_Last_Correction
VAR
	fb		: AstroBROT.FB_RADEC2HADEC;
	fbFresh	: AstroBROT.FB_RADEC2HADEC;
END_VAR
TEST('RADEC2HADEC_Switching_Off_Does_Not_Keep_The_Last_Correction');
fb(jd := 2461300.75, ra := 83.63, dec := 22.01, lon := -16.5);
fb(jd := 2461300.75, ra := 83.63, dec := 22.01, lon := -16.5, precess := FALSE, nutate := FALSE, aberration := FALSE);
fbFresh(jd := 2461300.75, ra := 83.63, dec := 22.01, lon := -16.5, precess := FALSE, nutate := FALSE, aberration := FALSE);
CheckAngle(fbFresh.ha_out, fb.ha_out, 1.0E-12, 'ha');
CheckNear(fbFresh.dec_out, fb.dec_out, 1.0E-12, 'dec');
TEST_FINISHED();
END_METHOD

METHOD PRIVATE RADEC2HADEC_Cyclic_Calls_With_Inputs_Set_Once_Are_Stable
VAR
	fb		: AstroBROT.FB_RADEC2HADEC;
	fbRef	: AstroBROT.FB_RADEC2HADEC;
	i		: INT;
END_VAR
TEST('RADEC2HADEC_Cyclic_Calls_With_Inputs_Set_Once_Are_Stable');
fbRef(jd := 2461300.75, ra := 83.63, dec := 22.01, lon := -16.5);
fb.jd := 2461300.75;
fb.ra := 83.63;
fb.dec := 22.01;
fb.lon := -16.5;
FOR i := 1 TO 5 DO
	fb();
	CheckAngle(fbRef.ha_out, fb.ha_out, 1.0E-12, 'cyclic call ha');
	CheckNear(fbRef.dec_out, fb.dec_out, 1.0E-12, 'cyclic call dec');
END_FOR
CheckNear(83.63, fb.ra, 0.0, 'ra input untouched');
CheckNear(22.01, fb.dec, 0.0, 'dec input untouched');
TEST_FINISHED();
END_METHOD

METHOD PRIVATE HADEC2RADEC_All_Switches_Off_Only_Applies_Sidereal_Time
VAR
	fb		: AstroBROT.FB_HADEC2RADEC;
	fLast	: LREAL;
END_VAR
TEST('HADEC2RADEC_All_Switches_Off_Only_Applies_Sidereal_Time');
fLast := ApparentSidereal(2461300.75, -16.5);
fb(jd := 2461300.75, ha := 345.0, dec := 22.01, lon := -16.5, precess := FALSE, nutate := FALSE, aberration := FALSE);
CheckAngle(fLast - 345.0, fb.ra_out, 1.0E-9, 'ra = LAST - ha');
CheckNear(22.01, fb.dec_out, 0.0, 'dec unchanged');
TEST_FINISHED();
END_METHOD

METHOD PRIVATE HADEC2RADEC_Each_Switch_Applies_Exactly_One_Correction
VAR
	fbOff		: AstroBROT.FB_HADEC2RADEC;
	fbPre		: AstroBROT.FB_HADEC2RADEC;
	fbNut		: AstroBROT.FB_HADEC2RADEC;
	fbAbr		: AstroBROT.FB_HADEC2RADEC;
	fbPrecess	: AstroBROT.FB_PRECESS;
	nut			: AstroBROT.FB_CO_NUTATE;
	abr			: AstroBROT.FB_CO_ABERRATION;
END_VAR
TEST('HADEC2RADEC_Each_Switch_Applies_Exactly_One_Correction');
fbOff(jd := 2461300.75, ha := 345.0, dec := 22.01, lon := -16.5, precess := FALSE, nutate := FALSE, aberration := FALSE);
fbPre(jd := 2461300.75, ha := 345.0, dec := 22.01, lon := -16.5, precess := TRUE, nutate := FALSE, aberration := FALSE);
fbNut(jd := 2461300.75, ha := 345.0, dec := 22.01, lon := -16.5, precess := FALSE, nutate := TRUE, aberration := FALSE);
fbAbr(jd := 2461300.75, ha := 345.0, dec := 22.01, lon := -16.5, precess := FALSE, nutate := FALSE, aberration := TRUE);
// the corrections are looked up at the position without any correction, like the block does
fbPrecess(ra := fbOff.ra_out, dec := fbOff.dec_out, equinox1 := AstroBROT.JD2JEPOCH(jd := 2461300.75), equinox2 := 2000.0);
nut(jd := 2461300.75, ra := fbOff.ra_out, dec := fbOff.dec_out);
abr(jd := 2461300.75, ra := fbOff.ra_out, dec := fbOff.dec_out);
AssertTrue(Condition := ABS(fbPrecess.ra_precessed - fbOff.ra_out) > 1.0E-3, Message := 'precession is not negligible');
AssertTrue(Condition := ABS(nut.d_ra) > 1.0E-5, Message := 'nutation is not negligible');
AssertTrue(Condition := ABS(abr.d_ra) > 1.0E-5, Message := 'aberration is not negligible');
CheckAngle(fbPrecess.ra_precessed, fbPre.ra_out, 1.0E-9, 'precession only: ra');
CheckNear(fbPrecess.dec_precessed, fbPre.dec_out, 1.0E-9, 'precession only: dec');
CheckAngle(fbOff.ra_out - nut.d_ra, fbNut.ra_out, 1.0E-9, 'nutation only: ra');
CheckNear(fbOff.dec_out - nut.d_dec, fbNut.dec_out, 1.0E-9, 'nutation only: dec');
CheckAngle(fbOff.ra_out - abr.d_ra, fbAbr.ra_out, 1.0E-9, 'aberration only: ra');
CheckNear(fbOff.dec_out - abr.d_dec, fbAbr.dec_out, 1.0E-9, 'aberration only: dec');
TEST_FINISHED();
END_METHOD

METHOD PRIVATE HADEC2RADEC_Right_Ascension_Is_Wrapped_Without_Precession
VAR
	fbLow	: AstroBROT.FB_HADEC2RADEC;
	fbHigh	: AstroBROT.FB_HADEC2RADEC;
	fLast	: LREAL;
END_VAR
TEST('HADEC2RADEC_Right_Ascension_Is_Wrapped_Without_Precession');
// the uncorrected RA is 1E-6 deg above 0 or below 360, the nutation and aberration correction (several
// arcsec) moves it across the wrap in one of the two cases
fLast := ApparentSidereal(2461300.75, -16.5);
fbLow(jd := 2461300.75, ha := fLast - 1.0E-6, dec := 22.01, lon := -16.5, precess := FALSE);
fbHigh(jd := 2461300.75, ha := fLast + 1.0E-6, dec := 22.01, lon := -16.5, precess := FALSE);
AssertTrue(Condition := fbLow.ra_out >= 0.0 AND fbLow.ra_out < 360.0, Message := 'ra in [0, 360) above the wrap');
AssertTrue(Condition := fbHigh.ra_out >= 0.0 AND fbHigh.ra_out < 360.0, Message := 'ra in [0, 360) below the wrap');
CheckAngle(0.0, fbLow.ra_out, 0.1, 'ra is near 0 above the wrap');
CheckAngle(0.0, fbHigh.ra_out, 0.1, 'ra is near 0 below the wrap');
TEST_FINISHED();
END_METHOD

METHOD PRIVATE HADEC2RADEC_Switching_Off_Does_Not_Keep_The_Last_Correction
VAR
	fb		: AstroBROT.FB_HADEC2RADEC;
	fbFresh	: AstroBROT.FB_HADEC2RADEC;
END_VAR
TEST('HADEC2RADEC_Switching_Off_Does_Not_Keep_The_Last_Correction');
fb(jd := 2461300.75, ha := 345.0, dec := 22.01, lon := -16.5);
fb(jd := 2461300.75, ha := 345.0, dec := 22.01, lon := -16.5, precess := FALSE, nutate := FALSE, aberration := FALSE);
fbFresh(jd := 2461300.75, ha := 345.0, dec := 22.01, lon := -16.5, precess := FALSE, nutate := FALSE, aberration := FALSE);
CheckAngle(fbFresh.ra_out, fb.ra_out, 1.0E-12, 'ra');
CheckNear(fbFresh.dec_out, fb.dec_out, 1.0E-12, 'dec');
TEST_FINISHED();
END_METHOD

METHOD PRIVATE EQ2HOR_Is_The_Composition_Of_Its_Parts
VAR
	fbEq	: AstroBROT.FB_EQ2HOR;
	fbHd	: AstroBROT.FB_RADEC2HADEC;
	fbAz	: AstroBROT.FB_HADEC2ALTAZ;
	i		: INT;
	bOn		: BOOL;
	bWs		: BOOL;
END_VAR
TEST('EQ2HOR_Is_The_Composition_Of_Its_Parts');
// no refraction: FB_EQ2HOR = FB_RADEC2HADEC + FB_HADEC2ALTAZ, with and without the corrections and with ws
FOR i := 0 TO 3 DO
	bOn := (i MOD 2) = 0;
	bWs := i >= 2;
	fbEq(jd := 2461300.75, ra := 83.63, dec := 22.01, lon := -16.5, lat := 48.5, ws := bWs, precess := bOn, nutate := bOn, aberration := TRUE, refract := FALSE);
	fbHd(jd := 2461300.75, ra := 83.63, dec := 22.01, lon := -16.5, precess := bOn, nutate := bOn, aberration := TRUE);
	fbAz(ha := fbHd.ha_out, dec := fbHd.dec_out, lat := 48.5, WS := bWs);
	CheckNear(fbAz.alt, fbEq.alt, 1.0E-12, 'alt');
	CheckAngle(fbAz.az, fbEq.az, 1.0E-12, 'az');
	CheckAngle(fbHd.ha_out, fbEq.ha, 1.0E-12, 'ha');
END_FOR
TEST_FINISHED();
END_METHOD

METHOD PRIVATE HOR2EQ_Is_The_Composition_Of_Its_Parts
VAR
	fbHor	: AstroBROT.FB_HOR2EQ;
	fbAh	: AstroBROT.FB_ALTAZ2HADEC;
	fbRd	: AstroBROT.FB_HADEC2RADEC;
	i		: INT;
	bOn		: BOOL;
	bWs		: BOOL;
	fAz		: LREAL;
END_VAR
TEST('HOR2EQ_Is_The_Composition_Of_Its_Parts');
// no refraction: FB_HOR2EQ = FB_ALTAZ2HADEC + FB_HADEC2RADEC, with and without the corrections and with ws
FOR i := 0 TO 3 DO
	bOn := (i MOD 2) = 0;
	bWs := i >= 2;
	fbHor(alt := 40.0, az := 120.0, jd := 2461300.75, lat := 48.5, lon := -16.5, ws := bWs, precess := bOn, nutate := bOn, aberration := TRUE, refract := FALSE);
	fAz := 120.0;
	IF bWs THEN
		fAz := 120.0 - 180.0;
	END_IF
	fbAh(alt := 40.0, az := fAz, lat := 48.5);
	fbRd(jd := 2461300.75, ha := fbAh.ha, dec := fbAh.dec, lon := -16.5, precess := bOn, nutate := bOn, aberration := TRUE);
	CheckAngle(fbRd.ra_out, fbHor.ra, 1.0E-12, 'ra');
	CheckNear(fbRd.dec_out, fbHor.dec, 1.0E-12, 'dec');
	CheckAngle(fbAh.ha, fbHor.ha, 1.0E-12, 'ha');
END_FOR
TEST_FINISHED();
END_METHOD

END_FUNCTION_BLOCK

// ---- POUs/FB_JD2LST_Tests.TcPOU
// Tests for AstroBROT.JD2LST (Julian Date -> local sidereal time in degrees) with the dut1 input (issue #12).
//
// jd is UTC, dut1 is UT1-UTC in seconds. Golden values come from AstroBROT/testing/golden_astro.py (the Python
// port, validated against erfa gmst82 by check_time_precess.py), tolerance 1e-9 deg. TwinCAT functions have no
// optional inputs, so every call passes dut1 explicitly.
FUNCTION_BLOCK FB_JD2LST_Tests EXTENDS TcUnit.FB_TestSuite
VAR
END_VAR

Golden_Values();
Dut1_Zero_Is_UTC_As_UT1();
Dut1_Shifts_By_The_Sidereal_Rate();
Wraps_Around_360();
Dut1_Is_Added_To_The_Time_Argument();

METHOD PRIVATE CheckAngle
VAR_INPUT
	fExpected	: LREAL;
	fActual		: LREAL;
	fDelta		: LREAL;
	sName		: STRING(255);
END_VAR
VAR
	fDiff	: LREAL;
END_VAR
// angles in degrees, compared modulo 360 so that 359.9999999 and -1.0E-7 are equal
fDiff := fActual - fExpected;
WHILE fDiff > 180.0 DO fDiff := fDiff - 360.0; END_WHILE
WHILE fDiff < -180.0 DO fDiff := fDiff + 360.0; END_WHILE
AssertEquals_LREAL(Expected := 0.0, Actual := fDiff, Delta := fDelta, Message := sName);
END_METHOD

METHOD PRIVATE CheckNear
VAR_INPUT
	fExpected	: LREAL;
	fActual		: LREAL;
	fDelta		: LREAL;
	sName		: STRING(255);
END_VAR
AssertEquals_LREAL(Expected := fExpected, Actual := fActual, Delta := fDelta, Message := sName);
END_METHOD

METHOD PRIVATE Dut1_Is_Added_To_The_Time_Argument
VAR

END_VAR
TEST('Dut1_Is_Added_To_The_Time_Argument');
// the same UT1 reached two ways: jd + 0.5 s with dut1 = 0 is jd with dut1 = 0.5
CheckNear(AstroBROT.JD2LST(jd := 2461300.75 + 0.5 / 86400.0, lon := 9.945392608768366, dut1 := 0.0), AstroBROT.JD2LST(jd := 2461300.75, lon := 9.945392608768366, dut1 := 0.5), 1.0E-9, 'jd + 0.5 s = dut1 0.5');
TEST_FINISHED();
END_METHOD

METHOD PRIVATE Dut1_Shifts_By_The_Sidereal_Rate
VAR
	fRate	: LREAL;
	fBase	: LREAL;
END_VAR
TEST('Dut1_Shifts_By_The_Sidereal_Rate');
// 1 s of UT1 is 360.98564736629 / 86400 deg of sidereal time. jd + dut1 / 86400 is quantised to about 40 us
// (jd is ~2.5E6 days), i.e. up to 1.7E-7 deg, so the tolerance is 5E-7 deg (1.8 mas), far below the 3.8E-3 deg shift.
fRate := 360.98564736629 / 86400.0;
fBase := AstroBROT.JD2LST(jd := 2461300.75, lon := 0.0, dut1 := 0.0);
CheckNear(fBase + 0.9 * fRate, AstroBROT.JD2LST(jd := 2461300.75, lon := 0.0, dut1 := 0.9), 5.0E-7, '+0.9 s');
CheckNear(fBase - 0.9 * fRate, AstroBROT.JD2LST(jd := 2461300.75, lon := 0.0, dut1 := -0.9), 5.0E-7, '-0.9 s');
TEST_FINISHED();
END_METHOD

METHOD PRIVATE Dut1_Zero_Is_UTC_As_UT1
VAR

END_VAR
TEST('Dut1_Zero_Is_UTC_As_UT1');
// dut1 = 0 reproduces the sidereal time of the version without the input (checked against erfa gmst82)
CheckNear(86.18993972893804, AstroBROT.JD2LST(jd := 2461300.75, lon := 0.0, dut1 := 0.0), 1.0E-9, 'dut1 = 0');
TEST_FINISHED();
END_METHOD

METHOD PRIVATE Golden_Values
VAR

END_VAR
TEST('Golden_Values');
CheckNear(86.18993972893804, AstroBROT.JD2LST(jd := 2461300.75, lon := 0.0, dut1 := 0.0), 1.0E-9, '2026 lon 0 dut1 +0.0');
CheckNear(86.19370005978271, AstroBROT.JD2LST(jd := 2461300.75, lon := 0.0, dut1 := 0.9), 1.0E-9, '2026 lon 0 dut1 +0.9');
CheckNear(86.18617939809337, AstroBROT.JD2LST(jd := 2461300.75, lon := 0.0, dut1 := -0.9), 1.0E-9, '2026 lon 0 dut1 -0.9');
CheckNear(96.13533233758062, AstroBROT.JD2LST(jd := 2461300.75, lon := 9.945392608768366, dut1 := 0.0), 1.0E-9, '2026 lon 9.945 dut1 +0.0');
CheckNear(96.13909266842529, AstroBROT.JD2LST(jd := 2461300.75, lon := 9.945392608768366, dut1 := 0.9), 1.0E-9, '2026 lon 9.945 dut1 +0.9');
CheckNear(96.13157200673595, AstroBROT.JD2LST(jd := 2461300.75, lon := 9.945392608768366, dut1 := -0.9), 1.0E-9, '2026 lon 9.945 dut1 -0.9');
CheckNear(100.53762762364931, AstroBROT.JD2LST(jd := 2455197.5, lon := 0.0, dut1 := 0.0), 1.0E-9, '2010 lon 0 dut1 +0.0');
CheckNear(100.54138795426115, AstroBROT.JD2LST(jd := 2455197.5, lon := 0.0, dut1 := 0.9), 1.0E-9, '2010 lon 0 dut1 +0.9');
CheckNear(100.53386729280464, AstroBROT.JD2LST(jd := 2455197.5, lon := 0.0, dut1 := -0.9), 1.0E-9, '2010 lon 0 dut1 -0.9');
CheckNear(110.48302023252472, AstroBROT.JD2LST(jd := 2455197.5, lon := 9.945392608768366, dut1 := 0.0), 1.0E-9, '2010 lon 9.945 dut1 +0.0');
CheckNear(110.48678056313656, AstroBROT.JD2LST(jd := 2455197.5, lon := 9.945392608768366, dut1 := 0.9), 1.0E-9, '2010 lon 9.945 dut1 +0.9');
CheckNear(110.47925990168005, AstroBROT.JD2LST(jd := 2455197.5, lon := 9.945392608768366, dut1 := -0.9), 1.0E-9, '2010 lon 9.945 dut1 -0.9');
TEST_FINISHED();
END_METHOD

METHOD PRIVATE Wraps_Around_360
VAR

END_VAR
TEST('Wraps_Around_360');
// lon 273.808 puts the sidereal time just below 360 deg, +0.9 s carries it past 360 deg
CheckNear(359.99793972913176, AstroBROT.JD2LST(jd := 2461300.75, lon := 273.808, dut1 := 0.0), 1.0E-9, 'just below 360');
CheckNear(0.0017000599764287472, AstroBROT.JD2LST(jd := 2461300.75, lon := 273.808, dut1 := 0.9), 1.0E-9, 'wrapped to just above 0');
TEST_FINISHED();
END_METHOD

END_FUNCTION_BLOCK

// ---- POUs/FB_EQ2HOR_Tests.TcPOU
// Tests for AstroBROT.FB_EQ2HOR (equatorial J2000 -> apparent horizontal coordinates).
//
// Golden values come from AstroBROT/testing/golden_astro.py (the Python port, validated against erfa). The port
// reproduces the ST to about 1e-10 deg, the tolerance here is 1e-7 deg (0.36 mas). Three sites: Tenerife 2026
// (high in the sky), Tenerife at about 20 deg altitude (refraction) and a southern site in 2010.
//
// Besides the numbers the tests pin down that the block never modifies its inputs and keeps no state between
// calls (issue #8). MAIN of the library assigns every input on every call, which hides both problems.
FUNCTION_BLOCK FB_EQ2HOR_Tests EXTENDS TcUnit.FB_TestSuite
VAR
END_VAR

Golden_All_Corrections_Tenerife_2026();
Golden_All_Corrections_Tenerife_low();
Golden_All_Corrections_South_2010();
Golden_Nutation_And_Aberration_Switches();
Toggling_The_Switches_Keeps_No_Stale_Corrections();
Inputs_Are_Not_Modified();
Cyclic_Calls_With_Inputs_Set_Once_Are_Stable();
Refraction_Tenerife_low();
Refraction_South_2010();
Golden_Dut1_Tenerife_2026();
Golden_Dut1_Tenerife_low();
Golden_Dut1_South_2010();

METHOD PRIVATE CheckNear
VAR_INPUT
	fExpected	: LREAL;
	fActual		: LREAL;
	fDelta		: LREAL;
	sName		: STRING(255);
END_VAR
AssertEquals_LREAL(Expected := fExpected, Actual := fActual, Delta := fDelta, Message := sName);
END_METHOD

METHOD PRIVATE CheckAngle
VAR_INPUT
	fExpected	: LREAL;
	fActual		: LREAL;
	fDelta		: LREAL;
	sName		: STRING(255);
END_VAR
VAR
	fDiff	: LREAL;
END_VAR
// angles in degrees, compared modulo 360 so that 359.9999999 and -1.0E-7 are equal
fDiff := fActual - fExpected;
WHILE fDiff > 180.0 DO fDiff := fDiff - 360.0; END_WHILE
WHILE fDiff < -180.0 DO fDiff := fDiff + 360.0; END_WHILE
AssertEquals_LREAL(Expected := 0.0, Actual := fDiff, Delta := fDelta, Message := sName);
END_METHOD

METHOD PRIVATE Golden_All_Corrections_Tenerife_2026
VAR
	fb	: AstroBROT.FB_EQ2HOR;
END_VAR
TEST('Golden_All_Corrections_Tenerife_2026');
fb(ra := 83.63, dec := 22.01, jd := 2461300.75, lon := -16.5, lat := 28.3, refract := FALSE);
CheckNear(75.59846498223517, fb.alt, 1.0E-7, 'Tenerife_2026 alt');
CheckAngle(112.59057933299366, fb.az, 1.0E-7, 'Tenerife_2026 az');
TEST_FINISHED();
END_METHOD

METHOD PRIVATE Golden_All_Corrections_Tenerife_low
VAR
	fb	: AstroBROT.FB_EQ2HOR;
END_VAR
TEST('Golden_All_Corrections_Tenerife_low');
fb(ra := 130.0, dec := -10.0, jd := 2461300.75, lon := -16.5, lat := 28.3, refract := FALSE);
CheckNear(20.004849547711906, fb.alt, 1.0E-7, 'Tenerife_low alt');
CheckAngle(114.06814750558047, fb.az, 1.0E-7, 'Tenerife_low az');
TEST_FINISHED();
END_METHOD

METHOD PRIVATE Golden_All_Corrections_South_2010
VAR
	fb	: AstroBROT.FB_EQ2HOR;
END_VAR
TEST('Golden_All_Corrections_South_2010');
fb(ra := 312.5, dec := -47.3, jd := 2455197.5, lon := -70.7, lat := -30.2, refract := FALSE);
CheckNear(29.98028023128418, fb.alt, 1.0E-7, 'South_2010 alt');
CheckAngle(229.80793288979396, fb.az, 1.0E-7, 'South_2010 az');
TEST_FINISHED();
END_METHOD

METHOD PRIVATE Golden_Nutation_And_Aberration_Switches
VAR
	fb01	: AstroBROT.FB_EQ2HOR;
	fb10	: AstroBROT.FB_EQ2HOR;
	fb00	: AstroBROT.FB_EQ2HOR;
END_VAR
TEST('Golden_Nutation_And_Aberration_Switches');
// nutate = FALSE still uses d_psi for the sidereal time, only the RA/Dec correction is skipped
fb10(ra := 83.63, dec := 22.01, jd := 2461300.75, lon := -16.5, lat := 28.3, refract := FALSE, nutate := TRUE, aberration := FALSE);
CheckNear(75.59846841386083, fb10.alt, 1.0E-7, 'Tenerife_2026 nutate=1 aberration=0 alt');
CheckAngle(112.59118972427912, fb10.az, 1.0E-7, 'Tenerife_2026 nutate=1 aberration=0 az');
fb01(ra := 83.63, dec := 22.01, jd := 2461300.75, lon := -16.5, lat := 28.3, refract := FALSE, nutate := FALSE, aberration := TRUE);
CheckNear(75.59936757788323, fb01.alt, 1.0E-7, 'Tenerife_2026 nutate=0 aberration=1 alt');
CheckAngle(112.60350125711398, fb01.az, 1.0E-7, 'Tenerife_2026 nutate=0 aberration=1 az');
fb00(ra := 83.63, dec := 22.01, jd := 2461300.75, lon := -16.5, lat := 28.3, refract := FALSE, nutate := FALSE, aberration := FALSE);
CheckNear(75.59937097997194, fb00.alt, 1.0E-7, 'Tenerife_2026 nutate=0 aberration=0 alt');
CheckAngle(112.60411169109408, fb00.az, 1.0E-7, 'Tenerife_2026 nutate=0 aberration=0 az');
fb10(ra := 312.5, dec := -47.3, jd := 2455197.5, lon := -70.7, lat := -30.2, refract := FALSE, nutate := TRUE, aberration := FALSE);
CheckNear(29.98438866090121, fb10.alt, 1.0E-7, 'South_2010 nutate=1 aberration=0 alt');
CheckAngle(229.8121407986145, fb10.az, 1.0E-7, 'South_2010 nutate=1 aberration=0 az');
fb01(ra := 312.5, dec := -47.3, jd := 2455197.5, lon := -70.7, lat := -30.2, refract := FALSE, nutate := FALSE, aberration := TRUE);
CheckNear(29.976340392064657, fb01.alt, 1.0E-7, 'South_2010 nutate=0 aberration=1 alt');
CheckAngle(229.8060751934534, fb01.az, 1.0E-7, 'South_2010 nutate=0 aberration=1 az');
fb00(ra := 312.5, dec := -47.3, jd := 2455197.5, lon := -70.7, lat := -30.2, refract := FALSE, nutate := FALSE, aberration := FALSE);
CheckNear(29.980448533028405, fb00.alt, 1.0E-7, 'South_2010 nutate=0 aberration=0 alt');
CheckAngle(229.81028321929855, fb00.az, 1.0E-7, 'South_2010 nutate=0 aberration=0 az');
TEST_FINISHED();
END_METHOD

METHOD PRIVATE Toggling_The_Switches_Keeps_No_Stale_Corrections
VAR
	fb	: AstroBROT.FB_EQ2HOR;
END_VAR
TEST('Toggling_The_Switches_Keeps_No_Stale_Corrections');
// the block keeps its correction deltas between calls; switching a flag off must drop that correction
fb(ra := 83.63, dec := 22.01, jd := 2461300.75, lon := -16.5, lat := 28.3, refract := FALSE, nutate := TRUE, aberration := TRUE);
CheckNear(75.59846498223517, fb.alt, 1.0E-7, 'toggle nutate=1 aberration=1 alt');
CheckAngle(112.59057933299366, fb.az, 1.0E-7, 'toggle nutate=1 aberration=1 az');
fb(ra := 83.63, dec := 22.01, jd := 2461300.75, lon := -16.5, lat := 28.3, refract := FALSE, nutate := FALSE, aberration := TRUE);
CheckNear(75.59936757788323, fb.alt, 1.0E-7, 'toggle nutate=0 aberration=1 alt');
CheckAngle(112.60350125711398, fb.az, 1.0E-7, 'toggle nutate=0 aberration=1 az');
fb(ra := 83.63, dec := 22.01, jd := 2461300.75, lon := -16.5, lat := 28.3, refract := FALSE, nutate := TRUE, aberration := FALSE);
CheckNear(75.59846841386083, fb.alt, 1.0E-7, 'toggle nutate=1 aberration=0 alt');
CheckAngle(112.59118972427912, fb.az, 1.0E-7, 'toggle nutate=1 aberration=0 az');
fb(ra := 83.63, dec := 22.01, jd := 2461300.75, lon := -16.5, lat := 28.3, refract := FALSE, nutate := FALSE, aberration := FALSE);
CheckNear(75.59937097997194, fb.alt, 1.0E-7, 'toggle nutate=0 aberration=0 alt');
CheckAngle(112.60411169109408, fb.az, 1.0E-7, 'toggle nutate=0 aberration=0 az');
fb(ra := 83.63, dec := 22.01, jd := 2461300.75, lon := -16.5, lat := 28.3, refract := FALSE, nutate := TRUE, aberration := TRUE);
CheckNear(75.59846498223517, fb.alt, 1.0E-7, 'toggle nutate=1 aberration=1 alt');
CheckAngle(112.59057933299366, fb.az, 1.0E-7, 'toggle nutate=1 aberration=1 az');
TEST_FINISHED();
END_METHOD

METHOD PRIVATE Inputs_Are_Not_Modified
VAR
	fb	: AstroBROT.FB_EQ2HOR;
END_VAR
TEST('Inputs_Are_Not_Modified');
fb(ra := 83.63, dec := 22.01, jd := 2461300.75, lon := -16.5, lat := 28.3, refract := TRUE);
CheckNear(83.63, fb.ra, 1.0E-15, 'ra unchanged');
CheckNear(22.01, fb.dec, 1.0E-15, 'dec unchanged');
CheckNear(2461300.75, fb.jd, 1.0E-15, 'jd unchanged');
TEST_FINISHED();
END_METHOD

METHOD PRIVATE Cyclic_Calls_With_Inputs_Set_Once_Are_Stable
VAR
	fb	: AstroBROT.FB_EQ2HOR;
	i	: INT;
END_VAR
TEST('Cyclic_Calls_With_Inputs_Set_Once_Are_Stable');
fb.ra := 83.63;
fb.dec := 22.01;
fb.jd := 2461300.75;
fb.lon := -16.5;
fb.lat := 28.3;
fb.refract := FALSE;
FOR i := 1 TO 5 DO
	// inputs are set once and the block is called cyclically, like a PLC program would do
	fb();
	CheckNear(75.59846498223517, fb.alt, 1.0E-7, 'cyclic call alt');
	CheckAngle(112.59057933299366, fb.az, 1.0E-7, 'cyclic call az');
END_FOR
TEST_FINISHED();
END_METHOD

METHOD PRIVATE Refraction_Tenerife_low
VAR
	fbObs	: AstroBROT.FB_EQ2HOR;
	fbGeo	: AstroBROT.FB_EQ2HOR;
END_VAR
TEST('Refraction_Tenerife_low');
fbObs(ra := 130.0, dec := -10.0, jd := 2461300.75, lon := -16.5, lat := 28.3, refract := TRUE, refract_to_observed := TRUE, altitude := 2400.0);
CheckNear(20.039496339721794, fbObs.alt, 1.0E-7, 'Tenerife_low to observed alt');
CheckAngle(114.06814750558047, fbObs.az, 1.0E-7, 'Tenerife_low to observed az');
fbGeo(ra := 130.0, dec := -10.0, jd := 2461300.75, lon := -16.5, lat := 28.3, refract := TRUE, refract_to_observed := FALSE, altitude := 2400.0);
CheckNear(19.970138517747017, fbGeo.alt, 1.0E-7, 'Tenerife_low to geometric alt');
CheckAngle(114.06814750558047, fbGeo.az, 1.0E-7, 'Tenerife_low to geometric az');
TEST_FINISHED();
END_METHOD

METHOD PRIVATE Refraction_South_2010
VAR
	fbObs	: AstroBROT.FB_EQ2HOR;
	fbGeo	: AstroBROT.FB_EQ2HOR;
END_VAR
TEST('Refraction_South_2010');
fbObs(ra := 312.5, dec := -47.3, jd := 2455197.5, lon := -70.7, lat := -30.2, refract := TRUE, refract_to_observed := TRUE, altitude := 2700.0);
CheckNear(30.001616325954682, fbObs.alt, 1.0E-7, 'South_2010 to observed alt');
CheckAngle(229.80793288979396, fbObs.az, 1.0E-7, 'South_2010 to observed az');
fbGeo(ra := 312.5, dec := -47.3, jd := 2455197.5, lon := -70.7, lat := -30.2, refract := TRUE, refract_to_observed := FALSE, altitude := 2700.0);
CheckNear(29.958925879892362, fbGeo.alt, 1.0E-7, 'South_2010 to geometric alt');
CheckAngle(229.80793288979396, fbGeo.az, 1.0E-7, 'South_2010 to geometric az');
TEST_FINISHED();
END_METHOD

METHOD PRIVATE Golden_Dut1_Tenerife_2026
VAR
	fb	: AstroBROT.FB_EQ2HOR;
END_VAR
TEST('Golden_Dut1_Tenerife_2026');
fb(ra := 83.63, dec := 22.01, jd := 2461300.75, lon := -16.5, lat := 28.3, refract := FALSE, dut1 := 0.9);
CheckNear(75.6015217605425, fb.alt, 1.0E-7, 'Tenerife_2026 dut1 +0.9 alt');
CheckAngle(112.59731630906032, fb.az, 1.0E-7, 'Tenerife_2026 dut1 +0.9 az');
fb(ra := 83.63, dec := 22.01, jd := 2461300.75, lon := -16.5, lat := 28.3, refract := FALSE, dut1 := -0.9);
CheckNear(75.5954080544077, fb.alt, 1.0E-7, 'Tenerife_2026 dut1 -0.9 alt');
CheckAngle(112.58384485334773, fb.az, 1.0E-7, 'Tenerife_2026 dut1 -0.9 az');
TEST_FINISHED();
END_METHOD

METHOD PRIVATE Golden_Dut1_Tenerife_low
VAR
	fb	: AstroBROT.FB_EQ2HOR;
END_VAR
TEST('Golden_Dut1_Tenerife_low');
fb(ra := 130.0, dec := -10.0, jd := 2461300.75, lon := -16.5, lat := 28.3, refract := FALSE, dut1 := 0.9);
CheckNear(20.007872562062794, fb.alt, 1.0E-7, 'Tenerife_low dut1 +0.9 alt');
CheckAngle(114.07042187844327, fb.az, 1.0E-7, 'Tenerife_low dut1 +0.9 az');
fb(ra := 130.0, dec := -10.0, jd := 2461300.75, lon := -16.5, lat := 28.3, refract := FALSE, dut1 := -0.9);
CheckNear(20.00182647976375, fb.alt, 1.0E-7, 'Tenerife_low dut1 -0.9 alt');
CheckAngle(114.06587325708954, fb.az, 1.0E-7, 'Tenerife_low dut1 -0.9 az');
TEST_FINISHED();
END_METHOD

METHOD PRIVATE Golden_Dut1_South_2010
VAR
	fb	: AstroBROT.FB_EQ2HOR;
END_VAR
TEST('Golden_Dut1_South_2010');
fb(ra := 312.5, dec := -47.3, jd := 2455197.5, lon := -70.7, lat := -30.2, refract := FALSE, dut1 := 0.9);
CheckNear(29.97779764757124, fb.alt, 1.0E-7, 'South_2010 dut1 +0.9 alt');
CheckAngle(229.80725126973925, fb.az, 1.0E-7, 'South_2010 dut1 +0.9 az');
fb(ra := 312.5, dec := -47.3, jd := 2455197.5, lon := -70.7, lat := -30.2, refract := FALSE, dut1 := -0.9);
CheckNear(29.982762840100285, fb.alt, 1.0E-7, 'South_2010 dut1 -0.9 alt');
CheckAngle(229.8086144058053, fb.az, 1.0E-7, 'South_2010 dut1 -0.9 az');
TEST_FINISHED();
END_METHOD

END_FUNCTION_BLOCK

// ---- POUs/FB_HOR2EQ_Tests.TcPOU
// Tests for AstroBROT.FB_HOR2EQ (horizontal -> equatorial J2000 coordinates).
//
// The alt/az inputs are fixed values (not the outputs of FB_EQ2HOR), so a shared error cannot cancel out. Golden
// values come from AstroBROT/testing/golden_astro.py, tolerance 1e-7 deg.
//
// The block must neither modify alt/az (the ws shift and the refraction correction used to be written back, issue
// #8) nor keep correction deltas between calls. MAIN of the library assigns every input on every call, which hides
// this, so the cyclic test sets the inputs once.
FUNCTION_BLOCK FB_HOR2EQ_Tests EXTENDS TcUnit.FB_TestSuite
VAR
END_VAR

Golden_All_Corrections_Tenerife_2026();
Golden_All_Corrections_Tenerife_low();
Golden_All_Corrections_South_2010();
Golden_Nutation_And_Aberration_Switches();
Toggling_The_Switches_Keeps_No_Stale_Corrections();
Azimuth_West_From_South();
Inputs_Are_Not_Modified();
Cyclic_Calls_With_Inputs_Set_Once_Are_Stable();
Refraction_Tenerife_low();
Refraction_South_2010();
Round_Trip_Through_FB_EQ2HOR();
Golden_Dut1_Tenerife_2026();
Golden_Dut1_Tenerife_low();
Golden_Dut1_South_2010();

METHOD PRIVATE CheckNear
VAR_INPUT
	fExpected	: LREAL;
	fActual		: LREAL;
	fDelta		: LREAL;
	sName		: STRING(255);
END_VAR
AssertEquals_LREAL(Expected := fExpected, Actual := fActual, Delta := fDelta, Message := sName);
END_METHOD

METHOD PRIVATE CheckAngle
VAR_INPUT
	fExpected	: LREAL;
	fActual		: LREAL;
	fDelta		: LREAL;
	sName		: STRING(255);
END_VAR
VAR
	fDiff	: LREAL;
END_VAR
// angles in degrees, compared modulo 360 so that 359.9999999 and -1.0E-7 are equal
fDiff := fActual - fExpected;
WHILE fDiff > 180.0 DO fDiff := fDiff - 360.0; END_WHILE
WHILE fDiff < -180.0 DO fDiff := fDiff + 360.0; END_WHILE
AssertEquals_LREAL(Expected := 0.0, Actual := fDiff, Delta := fDelta, Message := sName);
END_METHOD

METHOD PRIVATE Golden_All_Corrections_Tenerife_2026
VAR
	fb	: AstroBROT.FB_HOR2EQ;
END_VAR
TEST('Golden_All_Corrections_Tenerife_2026');
fb(alt := 52.0, az := 200.0, jd := 2461300.75, lon := -16.5, lat := 28.3, refract := FALSE);
CheckAngle(57.091388637043984, fb.ra, 1.0E-7, 'Tenerife_2026 ra');
CheckNear(-7.890511514810156, fb.dec, 1.0E-7, 'Tenerife_2026 dec');
TEST_FINISHED();
END_METHOD

METHOD PRIVATE Golden_All_Corrections_Tenerife_low
VAR
	fb	: AstroBROT.FB_HOR2EQ;
END_VAR
TEST('Golden_All_Corrections_Tenerife_low');
fb(alt := 21.0, az := 130.0, jd := 2461300.75, lon := -16.5, lat := 28.3, refract := FALSE);
CheckAngle(119.40414081413125, fb.ra, 1.0E-7, 'Tenerife_low ra');
CheckNear(-20.938138203483266, fb.dec, 1.0E-7, 'Tenerife_low dec');
TEST_FINISHED();
END_METHOD

METHOD PRIVATE Golden_All_Corrections_South_2010
VAR
	fb	: AstroBROT.FB_HOR2EQ;
END_VAR
TEST('Golden_All_Corrections_South_2010');
fb(alt := 63.5, az := 310.0, jd := 2455197.5, lon := -70.7, lat := -30.2, refract := FALSE);
CheckAngle(9.28374071008559, fb.ra, 1.0E-7, 'South_2010 ra');
CheckNear(-11.725986650809487, fb.dec, 1.0E-7, 'South_2010 dec');
TEST_FINISHED();
END_METHOD

METHOD PRIVATE Golden_Nutation_And_Aberration_Switches
VAR
	fb01	: AstroBROT.FB_HOR2EQ;
	fb10	: AstroBROT.FB_HOR2EQ;
	fb00	: AstroBROT.FB_HOR2EQ;
END_VAR
TEST('Golden_Nutation_And_Aberration_Switches');
fb10(alt := 52.0, az := 200.0, jd := 2461300.75, lon := -16.5, lat := 28.3, refract := FALSE, nutate := TRUE, aberration := FALSE);
CheckAngle(57.09380162014447, fb10.ra, 1.0E-7, 'Tenerife_2026 nutate=1 aberration=0 ra');
CheckNear(-7.88765562476953, fb10.dec, 1.0E-7, 'Tenerife_2026 nutate=1 aberration=0 dec');
fb01(alt := 52.0, az := 200.0, jd := 2461300.75, lon := -16.5, lat := 28.3, refract := FALSE, nutate := FALSE, aberration := TRUE);
CheckAngle(57.093669663716454, fb01.ra, 1.0E-7, 'Tenerife_2026 nutate=0 aberration=1 ra');
CheckNear(-7.8880514031941455, fb01.dec, 1.0E-7, 'Tenerife_2026 nutate=0 aberration=1 dec');
fb00(alt := 52.0, az := 200.0, jd := 2461300.75, lon := -16.5, lat := 28.3, refract := FALSE, nutate := FALSE, aberration := FALSE);
CheckAngle(57.096082646551956, fb00.ra, 1.0E-7, 'Tenerife_2026 nutate=0 aberration=0 ra');
CheckNear(-7.885195513018657, fb00.dec, 1.0E-7, 'Tenerife_2026 nutate=0 aberration=0 dec');
fb10(alt := 63.5, az := 310.0, jd := 2455197.5, lon := -70.7, lat := -30.2, refract := FALSE, nutate := TRUE, aberration := FALSE);
CheckAngle(9.283717099537949, fb10.ra, 1.0E-7, 'South_2010 nutate=1 aberration=0 ra');
CheckNear(-11.727565158724389, fb10.dec, 1.0E-7, 'South_2010 nutate=1 aberration=0 dec');
fb01(alt := 63.5, az := 310.0, jd := 2455197.5, lon := -70.7, lat := -30.2, refract := FALSE, nutate := FALSE, aberration := TRUE);
CheckAngle(9.288020281756417, fb01.ra, 1.0E-7, 'South_2010 nutate=0 aberration=1 ra');
CheckNear(-11.724069828122222, fb01.dec, 1.0E-7, 'South_2010 nutate=0 aberration=1 dec');
fb00(alt := 63.5, az := 310.0, jd := 2455197.5, lon := -70.7, lat := -30.2, refract := FALSE, nutate := FALSE, aberration := FALSE);
CheckAngle(9.287996671323913, fb00.ra, 1.0E-7, 'South_2010 nutate=0 aberration=0 ra');
CheckNear(-11.725648336038814, fb00.dec, 1.0E-7, 'South_2010 nutate=0 aberration=0 dec');
TEST_FINISHED();
END_METHOD

METHOD PRIVATE Toggling_The_Switches_Keeps_No_Stale_Corrections
VAR
	fb	: AstroBROT.FB_HOR2EQ;
END_VAR
TEST('Toggling_The_Switches_Keeps_No_Stale_Corrections');
// the block keeps its correction deltas between calls; switching a flag off must drop that correction
fb(alt := 52.0, az := 200.0, jd := 2461300.75, lon := -16.5, lat := 28.3, refract := FALSE, nutate := TRUE, aberration := TRUE);
CheckAngle(57.091388637043984, fb.ra, 1.0E-7, 'toggle nutate=1 aberration=1 ra');
CheckNear(-7.890511514810156, fb.dec, 1.0E-7, 'toggle nutate=1 aberration=1 dec');
fb(alt := 52.0, az := 200.0, jd := 2461300.75, lon := -16.5, lat := 28.3, refract := FALSE, nutate := FALSE, aberration := TRUE);
CheckAngle(57.093669663716454, fb.ra, 1.0E-7, 'toggle nutate=0 aberration=1 ra');
CheckNear(-7.8880514031941455, fb.dec, 1.0E-7, 'toggle nutate=0 aberration=1 dec');
fb(alt := 52.0, az := 200.0, jd := 2461300.75, lon := -16.5, lat := 28.3, refract := FALSE, nutate := TRUE, aberration := FALSE);
CheckAngle(57.09380162014447, fb.ra, 1.0E-7, 'toggle nutate=1 aberration=0 ra');
CheckNear(-7.88765562476953, fb.dec, 1.0E-7, 'toggle nutate=1 aberration=0 dec');
fb(alt := 52.0, az := 200.0, jd := 2461300.75, lon := -16.5, lat := 28.3, refract := FALSE, nutate := FALSE, aberration := FALSE);
CheckAngle(57.096082646551956, fb.ra, 1.0E-7, 'toggle nutate=0 aberration=0 ra');
CheckNear(-7.885195513018657, fb.dec, 1.0E-7, 'toggle nutate=0 aberration=0 dec');
fb(alt := 52.0, az := 200.0, jd := 2461300.75, lon := -16.5, lat := 28.3, refract := FALSE, nutate := TRUE, aberration := TRUE);
CheckAngle(57.091388637043984, fb.ra, 1.0E-7, 'toggle nutate=1 aberration=1 ra');
CheckNear(-7.890511514810156, fb.dec, 1.0E-7, 'toggle nutate=1 aberration=1 dec');
TEST_FINISHED();
END_METHOD

METHOD PRIVATE Azimuth_West_From_South
VAR
	fb	: AstroBROT.FB_HOR2EQ;
END_VAR
TEST('Azimuth_West_From_South');
fb(alt := 52.0, az := 200.0, jd := 2461300.75, lon := -16.5, lat := 28.3, refract := FALSE, ws := TRUE);
CheckAngle(95.72108173532322, fb.ra, 1.0E-7, 'ws = TRUE ra');
CheckNear(62.01980165070497, fb.dec, 1.0E-7, 'ws = TRUE dec');
TEST_FINISHED();
END_METHOD

METHOD PRIVATE Inputs_Are_Not_Modified
VAR
	fb	: AstroBROT.FB_HOR2EQ;
END_VAR
TEST('Inputs_Are_Not_Modified');
fb(alt := 52.0, az := 200.0, jd := 2461300.75, lon := -16.5, lat := 28.3, ws := TRUE, refract := TRUE, altitude := 2400.0);
CheckNear(52.0, fb.alt, 1.0E-15, 'alt unchanged (refraction is applied to a copy)');
CheckNear(200.0, fb.az, 1.0E-15, 'az unchanged (ws shift is applied to a copy)');
TEST_FINISHED();
END_METHOD

METHOD PRIVATE Cyclic_Calls_With_Inputs_Set_Once_Are_Stable
VAR
	fb	: AstroBROT.FB_HOR2EQ;
	i	: INT;
END_VAR
TEST('Cyclic_Calls_With_Inputs_Set_Once_Are_Stable');
fb.alt := 52.0;
fb.az := 200.0;
fb.jd := 2461300.75;
fb.lon := -16.5;
fb.lat := 28.3;
fb.ws := TRUE;
fb.refract := TRUE;
fb.altitude := 2400.0;
FOR i := 1 TO 5 DO
	// inputs are set once and the block is called cyclically; ws and refraction used to accumulate
	fb();
	CheckAngle(95.73459822152847, fb.ra, 1.0E-7, 'cyclic call, ws and refraction ra');
	CheckNear(62.02746769204616, fb.dec, 1.0E-7, 'cyclic call, ws and refraction dec');
END_FOR
TEST_FINISHED();
END_METHOD

METHOD PRIVATE Refraction_Tenerife_low
VAR
	fbObs	: AstroBROT.FB_HOR2EQ;
	fbGeo	: AstroBROT.FB_HOR2EQ;
END_VAR
TEST('Refraction_Tenerife_low');
fbObs(alt := 21.0, az := 130.0, jd := 2461300.75, lon := -16.5, lat := 28.3, refract := TRUE, alt_is_observed := TRUE, altitude := 2400.0);
CheckAngle(119.42969440304812, fbObs.ra, 1.0E-7, 'Tenerife_low alt is observed ra');
CheckNear(-20.96085779496941, fbObs.dec, 1.0E-7, 'Tenerife_low alt is observed dec');
fbGeo(alt := 21.0, az := 130.0, jd := 2461300.75, lon := -16.5, lat := 28.3, refract := TRUE, alt_is_observed := FALSE, altitude := 2400.0);
CheckAngle(119.37863816777192, fbGeo.ra, 1.0E-7, 'Tenerife_low alt is geometric ra');
CheckNear(-20.9154532358198, fbGeo.dec, 1.0E-7, 'Tenerife_low alt is geometric dec');
TEST_FINISHED();
END_METHOD

METHOD PRIVATE Refraction_South_2010
VAR
	fbObs	: AstroBROT.FB_HOR2EQ;
	fbGeo	: AstroBROT.FB_HOR2EQ;
END_VAR
TEST('Refraction_South_2010');
fbObs(alt := 63.5, az := 310.0, jd := 2455197.5, lon := -70.7, lat := -30.2, refract := TRUE, alt_is_observed := TRUE, altitude := 2700.0);
CheckAngle(9.279487019808851, fbObs.ra, 1.0E-7, 'South_2010 alt is observed ra');
CheckNear(-11.721448405755387, fbObs.dec, 1.0E-7, 'South_2010 alt is observed dec');
fbGeo(alt := 63.5, az := 310.0, jd := 2455197.5, lon := -70.7, lat := -30.2, refract := TRUE, alt_is_observed := FALSE, altitude := 2700.0);
CheckAngle(9.28799339553679, fbGeo.ra, 1.0E-7, 'South_2010 alt is geometric ra');
CheckNear(-11.730523611820027, fbGeo.dec, 1.0E-7, 'South_2010 alt is geometric dec');
TEST_FINISHED();
END_METHOD

METHOD PRIVATE Round_Trip_Through_FB_EQ2HOR
VAR
	fbEq	: AstroBROT.FB_EQ2HOR;
	fbHor	: AstroBROT.FB_HOR2EQ;
END_VAR
TEST('Round_Trip_Through_FB_EQ2HOR');
// the two blocks apply nutation and aberration at slightly different positions, so they are only approximate
// inverses: the round trip is off by up to 0.34 mas (3.4E-7 deg, same in the Python port), hence the wider tolerance
fbEq(ra := 83.63, dec := 22.01, jd := 2461300.75, lon := -16.5, lat := 28.3, refract := FALSE);
fbHor(alt := fbEq.alt, az := fbEq.az, jd := 2461300.75, lon := -16.5, lat := 28.3, refract := FALSE);
CheckAngle(83.63, fbHor.ra, 1.0E-6, 'Tenerife_2026 ra round trip');
CheckNear(22.01, fbHor.dec, 1.0E-6, 'Tenerife_2026 dec round trip');
fbEq(ra := 130.0, dec := -10.0, jd := 2461300.75, lon := -16.5, lat := 28.3, refract := FALSE);
fbHor(alt := fbEq.alt, az := fbEq.az, jd := 2461300.75, lon := -16.5, lat := 28.3, refract := FALSE);
CheckAngle(130.0, fbHor.ra, 1.0E-6, 'Tenerife_low ra round trip');
CheckNear(-10.0, fbHor.dec, 1.0E-6, 'Tenerife_low dec round trip');
fbEq(ra := 312.5, dec := -47.3, jd := 2455197.5, lon := -70.7, lat := -30.2, refract := FALSE);
fbHor(alt := fbEq.alt, az := fbEq.az, jd := 2455197.5, lon := -70.7, lat := -30.2, refract := FALSE);
CheckAngle(312.5, fbHor.ra, 1.0E-6, 'South_2010 ra round trip');
CheckNear(-47.3, fbHor.dec, 1.0E-6, 'South_2010 dec round trip');
TEST_FINISHED();
END_METHOD

METHOD PRIVATE Golden_Dut1_Tenerife_2026
VAR
	fb	: AstroBROT.FB_HOR2EQ;
END_VAR
TEST('Golden_Dut1_Tenerife_2026');
fb(alt := 52.0, az := 200.0, jd := 2461300.75, lat := 28.3, lon := -16.5, refract := FALSE, dut1 := 0.9);
CheckAngle(57.09515001446652, fb.ra, 1.0E-7, 'Tenerife_2026 dut1 +0.9 ra');
CheckNear(-7.890503354473438, fb.dec, 1.0E-7, 'Tenerife_2026 dut1 +0.9 dec');
fb(alt := 52.0, az := 200.0, jd := 2461300.75, lat := 28.3, lon := -16.5, refract := FALSE, dut1 := -0.9);
CheckAngle(57.08762725955663, fb.ra, 1.0E-7, 'Tenerife_2026 dut1 -0.9 ra');
CheckNear(-7.890519674787103, fb.dec, 1.0E-7, 'Tenerife_2026 dut1 -0.9 dec');
TEST_FINISHED();
END_METHOD

METHOD PRIVATE Golden_Dut1_Tenerife_low
VAR
	fb	: AstroBROT.FB_HOR2EQ;
END_VAR
TEST('Golden_Dut1_Tenerife_low');
fb(alt := 21.0, az := 130.0, jd := 2461300.75, lat := 28.3, lon := -16.5, refract := FALSE, dut1 := 0.9);
CheckAngle(119.4078996268092, fb.ra, 1.0E-7, 'Tenerife_low dut1 +0.9 ra');
CheckNear(-20.938129516273722, fb.dec, 1.0E-7, 'Tenerife_low dut1 +0.9 dec');
fb(alt := 21.0, az := 130.0, jd := 2461300.75, lat := 28.3, lon := -16.5, refract := FALSE, dut1 := -0.9);
CheckAngle(119.40038200122402, fb.ra, 1.0E-7, 'Tenerife_low dut1 -0.9 ra');
CheckNear(-20.938146890995743, fb.dec, 1.0E-7, 'Tenerife_low dut1 -0.9 dec');
TEST_FINISHED();
END_METHOD

METHOD PRIVATE Golden_Dut1_South_2010
VAR
	fb	: AstroBROT.FB_HOR2EQ;
END_VAR
TEST('Golden_Dut1_South_2010');
fb(alt := 63.5, az := 310.0, jd := 2455197.5, lat := -30.2, lon := -70.7, refract := FALSE, dut1 := 0.9);
CheckAngle(9.287501426247882, fb.ra, 1.0E-7, 'South_2010 dut1 +0.9 ra');
CheckNear(-11.725986088100136, fb.dec, 1.0E-7, 'South_2010 dut1 +0.9 dec');
fb(alt := 63.5, az := 310.0, jd := 2455197.5, lat := -30.2, lon := -70.7, refract := FALSE, dut1 := -0.9);
CheckAngle(9.27997999368262, fb.ra, 1.0E-7, 'South_2010 dut1 -0.9 ra');
CheckNear(-11.725987213279037, fb.dec, 1.0E-7, 'South_2010 dut1 -0.9 dec');
TEST_FINISHED();
END_METHOD

END_FUNCTION_BLOCK

// ---- POUs/FB_TEN_Tests.TcPOU
// Tests for AstroBROT.TEN (sexagesimal to decimal).
//
// Sign convention of IDLAstro's ten: a minus sign on any nonzero element makes the whole value negative, so
// TEN(-5, 30, 0) = -5.5 and TEN(0, -23, 34) = -0.39277778 (the example from the IDL documentation), tolerance 1e-12.
FUNCTION_BLOCK FB_TEN_Tests EXTENDS TcUnit.FB_TestSuite
VAR
END_VAR

Positive_Values();
Negative_Degrees_Apply_To_The_Whole_Value();
Negative_Minutes_Or_Seconds_Apply_To_The_Whole_Value();
Zero_Is_Zero();

METHOD PRIVATE CheckNear
VAR_INPUT
	fExpected	: LREAL;
	fActual		: LREAL;
	fDelta		: LREAL;
	sName		: STRING(255);
END_VAR
AssertEquals_LREAL(Expected := fExpected, Actual := fActual, Delta := fDelta, Message := sName);
END_METHOD

METHOD PRIVATE Positive_Values
VAR
END_VAR
TEST('Positive_Values');
CheckNear(5.5, AstroBROT.TEN(5.0, 30.0, 0.0), 1.0E-12, 'TEN(5, 30, 0)');
CheckNear(10.392777777777777, AstroBROT.TEN(10.0, 23.0, 34.0), 1.0E-12, 'TEN(10, 23, 34)');
TEST_FINISHED();
END_METHOD

METHOD PRIVATE Negative_Degrees_Apply_To_The_Whole_Value
VAR
END_VAR
TEST('Negative_Degrees_Apply_To_The_Whole_Value');
CheckNear(-5.5, AstroBROT.TEN(-5.0, 30.0, 0.0), 1.0E-12, 'TEN(-5, 30, 0)');
CheckNear(-1.0341666666666667, AstroBROT.TEN(-1.0, 2.0, 3.0), 1.0E-12, 'TEN(-1, 2, 3)');
TEST_FINISHED();
END_METHOD

METHOD PRIVATE Negative_Minutes_Or_Seconds_Apply_To_The_Whole_Value
VAR
END_VAR
TEST('Negative_Minutes_Or_Seconds_Apply_To_The_Whole_Value');
CheckNear(-0.3927777777777778, AstroBROT.TEN(0.0, -23.0, 34.0), 1.0E-12, 'TEN(0, -23, 34)');
CheckNear(-5.5, AstroBROT.TEN(5.0, -30.0, 0.0), 1.0E-12, 'TEN(5, -30, 0)');
CheckNear(-1.0341666666666667, AstroBROT.TEN(1.0, 2.0, -3.0), 1.0E-12, 'TEN(1, 2, -3)');
CheckNear(-0.008333333333333333, AstroBROT.TEN(0.0, 0.0, -30.0), 1.0E-12, 'TEN(0, 0, -30)');
TEST_FINISHED();
END_METHOD

METHOD PRIVATE Zero_Is_Zero
VAR
END_VAR
TEST('Zero_Is_Zero');
CheckNear(0.0, AstroBROT.TEN(0.0, 0.0, 0.0), 1.0E-15, 'TEN(0, 0, 0)');
TEST_FINISHED();
END_METHOD

END_FUNCTION_BLOCK

// ---- POUs/FB_PRECESS_Tests.TcPOU
// Tests for AstroBROT.FB_PRECESS (P03 precession between two Julian epochs, via J2000).
//
// GENERATED by AstroBROT/testing/gen_block_tests.py from testing/golden_blocks.py, do not edit the numbers by hand.
// Every golden case is checked twice: against the Python port of the ST (tolerance 1E-8 deg, catches any change of
// behaviour) and against erfa.bp06 (precession matrix, great-circle separation 1E-5 deg = 0.036 arcsec, catches an
// error the port shares with the ST). The relation tests do not need golden values at all.
//
// FB_PRECESS only rotates between J2000 and one other epoch, so a general epoch pair goes through J2000 (issue #9).
FUNCTION_BLOCK FB_PRECESS_Tests EXTENDS TcUnit.FB_TestSuite
VAR
END_VAR

Golden_J2000_To_Date();
Golden_Between_Two_Epochs();
Golden_RA_Wrap();
Golden_Poles();
Same_Epoch_Is_Identity();
Round_Trip_Through_J2000();
Two_Steps_Equal_Precessing_Via_J2000();
Right_Ascension_Is_Normalised();
Inputs_Are_Not_Modified();
Cyclic_Calls_With_Inputs_Set_Once_Are_Stable();

METHOD PRIVATE CheckNear
VAR_INPUT
	fExpected	: LREAL;
	fActual	: LREAL;
	fDelta	: LREAL;
	sName	: STRING(255);
END_VAR
AssertEquals_LREAL(Expected := fExpected, Actual := fActual, Delta := fDelta, Message := sName);
END_METHOD

METHOD PRIVATE CheckAngle
VAR_INPUT
	fExpected	: LREAL;
	fActual	: LREAL;
	fDelta	: LREAL;
	sName	: STRING(255);
END_VAR
VAR
	fDiff	: LREAL;
END_VAR
// angles in degrees, compared modulo 360 so that 359.9999999 and -1.0E-7 are equal
fDiff := fActual - fExpected;
WHILE fDiff > 180.0 DO fDiff := fDiff - 360.0; END_WHILE
WHILE fDiff < -180.0 DO fDiff := fDiff + 360.0; END_WHILE
AssertEquals_LREAL(Expected := 0.0, Actual := fDiff, Delta := fDelta, Message := sName);
END_METHOD

METHOD PRIVATE CheckSeparation
VAR_INPUT
	fLon1	: LREAL;
	fLat1	: LREAL;
	fLon2	: LREAL;
	fLat2	: LREAL;
	fDelta	: LREAL;
	sName	: STRING(255);
END_VAR
VAR
	fD2r	: LREAL;
	fHalfDLat	: LREAL;
	fHalfDLon	: LREAL;
	fHav	: LREAL;
	fSep	: LREAL;
END_VAR
// great-circle separation of two positions (longitude, latitude in degrees) against a tolerance in degrees;
// a difference of longitudes is not a distance on the sky, this is (haversine formula)
fD2r := 0.017453292519943295;
fHalfDLat := (fLat2 - fLat1) * fD2r * 0.5;
fHalfDLon := (fLon2 - fLon1) * fD2r * 0.5;
fHav := SIN(fHalfDLat) * SIN(fHalfDLat) + COS(fLat1 * fD2r) * COS(fLat2 * fD2r) * SIN(fHalfDLon) * SIN(fHalfDLon);
fSep := 2.0 * ASIN(SQRT(LIMIT(0.0, fHav, 1.0))) / fD2r;
AssertEquals_LREAL(Expected := 0.0, Actual := fSep, Delta := fDelta, Message := sName);
END_METHOD

METHOD PRIVATE Golden_J2000_To_Date
VAR
	fb	: AstroBROT.FB_PRECESS;
END_VAR
TEST('Golden_J2000_To_Date');
fb(ra := 83.63, dec := 22.01, equinox1 := 2000.0, equinox2 := 2026.5);
CheckAngle(84.02884460749144, fb.ra_precessed, 1.0E-8, 'J2000_to_2026 ra');
CheckNear(22.0258551337181, fb.dec_precessed, 1.0E-8, 'J2000_to_2026 dec');
CheckSeparation(84.02884460749591, 22.025855133729486, fb.ra_precessed, fb.dec_precessed, 1.0E-5, 'J2000_to_2026 vs erfa');
fb(ra := 312.5, dec := -47.3, equinox1 := 2000.0, equinox2 := 2010.0);
CheckAngle(312.6725080638107, fb.ra_precessed, 1.0E-8, 'J2000_to_2010_south ra');
CheckNear(-47.262327080321406, fb.dec_precessed, 1.0E-8, 'J2000_to_2010_south dec');
CheckSeparation(312.6725080638149, -47.26232708032657, fb.ra_precessed, fb.dec_precessed, 1.0E-5, 'J2000_to_2010_south vs erfa');
TEST_FINISHED();
END_METHOD

METHOD PRIVATE Golden_Between_Two_Epochs
VAR
	fb	: AstroBROT.FB_PRECESS;
END_VAR
TEST('Golden_Between_Two_Epochs');
fb(ra := 10.0, dec := 20.0, equinox1 := 2010.0, equinox2 := 2020.0);
CheckAngle(10.131674024998764, fb.ra_precessed, 1.0E-8, 'Both_epochs_not_J2000 ra');
CheckNear(20.054811409601943, fb.dec_precessed, 1.0E-8, 'Both_epochs_not_J2000 dec');
CheckSeparation(10.13167402499991, 20.05481140959979, fb.ra_precessed, fb.dec_precessed, 1.0E-5, 'Both_epochs_not_J2000 vs erfa');
fb(ra := 10.0, dec := 20.0, equinox1 := 2020.0, equinox2 := 2000.0);
CheckAngle(9.736828222801343, fb.ra_precessed, 1.0E-8, 'Back_to_J2000 ra');
CheckNear(19.890308491600006, fb.dec_precessed, 1.0E-8, 'Back_to_J2000 dec');
CheckSeparation(9.73682822279856, 19.890308491604287, fb.ra_precessed, fb.dec_precessed, 1.0E-5, 'Back_to_J2000 vs erfa');
fb(ra := 200.0, dec := -30.0, equinox1 := 1950.0, equinox2 := 2000.0);
CheckAngle(200.69666810482232, fb.ra_precessed, 1.0E-8, 'From_1950 ra');
CheckNear(-30.261014690476078, fb.dec_precessed, 1.0E-8, 'From_1950 dec');
CheckSeparation(200.69666810483287, -30.26101469046997, fb.ra_precessed, fb.dec_precessed, 1.0E-5, 'From_1950 vs erfa');
TEST_FINISHED();
END_METHOD

METHOD PRIVATE Golden_RA_Wrap
VAR
	fb	: AstroBROT.FB_PRECESS;
END_VAR
TEST('Golden_RA_Wrap');
fb(ra := 359.9999, dec := 10.0, equinox1 := 2000.0, equinox2 := 2050.0);
CheckAngle(0.6408546660457171, fb.ra_precessed, 1.0E-8, 'RA_wrap_up ra');
CheckNear(10.278324337869142, fb.dec_precessed, 1.0E-8, 'RA_wrap_up dec');
CheckSeparation(0.6408546660547558, 10.2783243378534, fb.ra_precessed, fb.dec_precessed, 1.0E-5, 'RA_wrap_up vs erfa');
fb(ra := 0.0001, dec := 10.0, equinox1 := 2000.0, equinox2 := 1950.0);
CheckAngle(359.3598872118728, fb.ra_precessed, 1.0E-8, 'RA_wrap_down ra');
CheckNear(9.721615962410127, fb.dec_precessed, 1.0E-8, 'RA_wrap_down dec');
CheckSeparation(359.35988721185373, 9.72161596242269, fb.ra_precessed, fb.dec_precessed, 1.0E-5, 'RA_wrap_down vs erfa');
TEST_FINISHED();
END_METHOD

METHOD PRIVATE Golden_Poles
VAR
	fb	: AstroBROT.FB_PRECESS;
END_VAR
TEST('Golden_Poles');
fb(ra := 0.0, dec := 90.0, equinox1 := 2000.0, equinox2 := 2030.0);
CheckAngle(180.19146429912647, fb.ra_precessed, 1.0E-8, 'North_pole ra');
CheckNear(89.83299505910631, fb.dec_precessed, 1.0E-8, 'North_pole dec');
CheckSeparation(180.1914643039869, 89.83299505911724, fb.ra_precessed, fb.dec_precessed, 1.0E-5, 'North_pole vs erfa');
fb(ra := 0.0, dec := -90.0, equinox1 := 2000.0, equinox2 := 2030.0);
CheckAngle(0.1914642991264698, fb.ra_precessed, 1.0E-8, 'South_pole ra');
CheckNear(-89.83299505910631, fb.dec_precessed, 1.0E-8, 'South_pole dec');
CheckSeparation(0.19146430398690156, -89.83299505911724, fb.ra_precessed, fb.dec_precessed, 1.0E-5, 'South_pole vs erfa');
TEST_FINISHED();
END_METHOD

METHOD PRIVATE Same_Epoch_Is_Identity
VAR
	fb	: AstroBROT.FB_PRECESS;
END_VAR
TEST('Same_Epoch_Is_Identity');
fb(ra := 123.4, dec := -56.7, equinox1 := 2015.0, equinox2 := 2015.0);
CheckAngle(123.4, fb.ra_precessed, 1.0E-12, 'ra');
CheckNear(-56.7, fb.dec_precessed, 1.0E-12, 'dec');
fb(ra := 123.4, dec := -56.7, equinox1 := 2000.0, equinox2 := 2000.0);
CheckAngle(123.4, fb.ra_precessed, 1.0E-12, 'J2000 ra');
CheckNear(-56.7, fb.dec_precessed, 1.0E-12, 'J2000 dec');
TEST_FINISHED();
END_METHOD

METHOD PRIVATE Round_Trip_Through_J2000
VAR
	fb	: AstroBROT.FB_PRECESS;
	fbBack	: AstroBROT.FB_PRECESS;
END_VAR
TEST('Round_Trip_Through_J2000');
fb(ra := 83.63, dec := 22.01, equinox1 := 2000.0, equinox2 := 2050.0);
fbBack(ra := fb.ra_precessed, dec := fb.dec_precessed, equinox1 := 2050.0, equinox2 := 2000.0);
CheckAngle(83.63, fbBack.ra_precessed, 1.0E-9, 'J2000 -> 2050 -> J2000 ra');
CheckNear(22.01, fbBack.dec_precessed, 1.0E-9, 'J2000 -> 2050 -> J2000 dec');
fb(ra := 10.0, dec := 20.0, equinox1 := 2010.0, equinox2 := 2030.0);
fbBack(ra := fb.ra_precessed, dec := fb.dec_precessed, equinox1 := 2030.0, equinox2 := 2010.0);
CheckAngle(10.0, fbBack.ra_precessed, 1.0E-9, '2010 -> 2030 -> 2010 ra');
CheckNear(20.0, fbBack.dec_precessed, 1.0E-9, '2010 -> 2030 -> 2010 dec');
TEST_FINISHED();
END_METHOD

METHOD PRIVATE Two_Steps_Equal_Precessing_Via_J2000
VAR
	fb	: AstroBROT.FB_PRECESS;
	fbA	: AstroBROT.FB_PRECESS;
	fbB	: AstroBROT.FB_PRECESS;
END_VAR
TEST('Two_Steps_Equal_Precessing_Via_J2000');
// before the fix of issue #9 a step between two epochs that are both not J2000 gave the wrong result
fb(ra := 10.0, dec := 20.0, equinox1 := 2010.0, equinox2 := 2020.0);
fbA(ra := 10.0, dec := 20.0, equinox1 := 2010.0, equinox2 := 2000.0);
fbB(ra := fbA.ra_precessed, dec := fbA.dec_precessed, equinox1 := 2000.0, equinox2 := 2020.0);
CheckAngle(fbB.ra_precessed, fb.ra_precessed, 1.0E-9, 'ra');
CheckNear(fbB.dec_precessed, fb.dec_precessed, 1.0E-9, 'dec');
// and 2010 -> 2020 is not the same rotation as 2000 -> 2010
fbA(ra := 10.0, dec := 20.0, equinox1 := 2000.0, equinox2 := 2010.0);
AssertTrue(Condition := ABS(fb.ra_precessed - fbA.ra_precessed) > 1.0E-6, Message := 'shifted epochs give a different result');
TEST_FINISHED();
END_METHOD

METHOD PRIVATE Right_Ascension_Is_Normalised
VAR
	fb	: AstroBROT.FB_PRECESS;
	fbRef	: AstroBROT.FB_PRECESS;
	fbShift	: AstroBROT.FB_PRECESS;
END_VAR
TEST('Right_Ascension_Is_Normalised');
fbRef(ra := 350.0, dec := -40.0, equinox1 := 2000.0, equinox2 := 2030.0);
fb(ra := -10.0, dec := -40.0, equinox1 := 2000.0, equinox2 := 2030.0);
CheckAngle(fbRef.ra_precessed, fb.ra_precessed, 1.0E-9, 'ra -10 is 350');
AssertTrue(Condition := fb.ra_precessed >= 0.0 AND fb.ra_precessed < 360.0, Message := 'ra -10 gives 0 <= ra < 360');
fbShift(ra := 710.0, dec := -40.0, equinox1 := 2000.0, equinox2 := 2030.0);
CheckAngle(fbRef.ra_precessed, fbShift.ra_precessed, 1.0E-9, 'ra 710 is 350');
AssertTrue(Condition := fbShift.ra_precessed >= 0.0 AND fbShift.ra_precessed < 360.0, Message := 'ra 710 gives 0 <= ra < 360');
TEST_FINISHED();
END_METHOD

METHOD PRIVATE Inputs_Are_Not_Modified
VAR
	fb	: AstroBROT.FB_PRECESS;
END_VAR
TEST('Inputs_Are_Not_Modified');
fb(ra := 83.63, dec := 22.01, equinox1 := 2000.0, equinox2 := 2026.5);
CheckNear(83.63, fb.ra, 1.0E-15, 'ra unchanged');
CheckNear(22.01, fb.dec, 1.0E-15, 'dec unchanged');
CheckNear(2000.0, fb.equinox1, 1.0E-15, 'equinox1 unchanged');
CheckNear(2026.5, fb.equinox2, 1.0E-15, 'equinox2 unchanged');
TEST_FINISHED();
END_METHOD

METHOD PRIVATE Cyclic_Calls_With_Inputs_Set_Once_Are_Stable
VAR
	fb	: AstroBROT.FB_PRECESS;
	i	: INT;
END_VAR
TEST('Cyclic_Calls_With_Inputs_Set_Once_Are_Stable');
fb.ra := 83.63;
fb.dec := 22.01;
fb.equinox1 := 2000.0;
fb.equinox2 := 2026.5;
FOR i := 1 TO 5 DO
	fb();
	CheckAngle(84.02884460749144, fb.ra_precessed, 1.0E-8, 'cyclic call ra');
	CheckNear(22.0258551337181, fb.dec_precessed, 1.0E-8, 'cyclic call dec');
END_FOR
TEST_FINISHED();
END_METHOD

END_FUNCTION_BLOCK

// ---- POUs/FB_RADEC2HADEC_Tests.TcPOU
// Tests for AstroBROT.FB_RADEC2HADEC (ICRS RA/Dec -> apparent hour angle / Dec; the block IAG50cm uses).
//
// GENERATED by AstroBROT/testing/gen_block_tests.py from testing/golden_blocks.py, do not edit the numbers by hand.
// Every golden case is checked against the Python port of the ST (1E-7 deg) and against erfa.atco13 as a great-circle
// separation on the (HA, Dec) sphere (2E-4 deg = 0.72 arcsec; the port is 0.2 to 0.4 arcsec away, mostly the diurnal
// aberration that the ST leaves out). The dut1 shift itself is also covered in FB_DUT1_Tests.
//
// Every call assigns all inputs: FB_RADEC2HADEC still writes its precessed and corrected position back into ra and dec
// (issue #8), so these tests must not rely on ra / dec surviving a call.
FUNCTION_BLOCK FB_RADEC2HADEC_Tests EXTENDS TcUnit.FB_TestSuite
VAR
END_VAR

Golden_Tenerife_2026();
Golden_Tenerife_low();
Golden_South_2010();
Golden_Dut1();
Golden_RA_Wrap();
Golden_Poles();
Golden_Near_The_Poles();
Right_Ascension_Is_Periodic();
Longitude_Is_Periodic();
Outputs_Stay_In_Range();
Time_Inputs_Are_Not_Modified();

METHOD PRIVATE CheckNear
VAR_INPUT
	fExpected	: LREAL;
	fActual	: LREAL;
	fDelta	: LREAL;
	sName	: STRING(255);
END_VAR
AssertEquals_LREAL(Expected := fExpected, Actual := fActual, Delta := fDelta, Message := sName);
END_METHOD

METHOD PRIVATE CheckAngle
VAR_INPUT
	fExpected	: LREAL;
	fActual	: LREAL;
	fDelta	: LREAL;
	sName	: STRING(255);
END_VAR
VAR
	fDiff	: LREAL;
END_VAR
// angles in degrees, compared modulo 360 so that 359.9999999 and -1.0E-7 are equal
fDiff := fActual - fExpected;
WHILE fDiff > 180.0 DO fDiff := fDiff - 360.0; END_WHILE
WHILE fDiff < -180.0 DO fDiff := fDiff + 360.0; END_WHILE
AssertEquals_LREAL(Expected := 0.0, Actual := fDiff, Delta := fDelta, Message := sName);
END_METHOD

METHOD PRIVATE CheckSeparation
VAR_INPUT
	fLon1	: LREAL;
	fLat1	: LREAL;
	fLon2	: LREAL;
	fLat2	: LREAL;
	fDelta	: LREAL;
	sName	: STRING(255);
END_VAR
VAR
	fD2r	: LREAL;
	fHalfDLat	: LREAL;
	fHalfDLon	: LREAL;
	fHav	: LREAL;
	fSep	: LREAL;
END_VAR
// great-circle separation of two positions (longitude, latitude in degrees) against a tolerance in degrees;
// a difference of longitudes is not a distance on the sky, this is (haversine formula)
fD2r := 0.017453292519943295;
fHalfDLat := (fLat2 - fLat1) * fD2r * 0.5;
fHalfDLon := (fLon2 - fLon1) * fD2r * 0.5;
fHav := SIN(fHalfDLat) * SIN(fHalfDLat) + COS(fLat1 * fD2r) * COS(fLat2 * fD2r) * SIN(fHalfDLon) * SIN(fHalfDLon);
fSep := 2.0 * ASIN(SQRT(LIMIT(0.0, fHav, 1.0))) / fD2r;
AssertEquals_LREAL(Expected := 0.0, Actual := fSep, Delta := fDelta, Message := sName);
END_METHOD

METHOD PRIVATE Golden_Tenerife_2026
VAR
	fb	: AstroBROT.FB_RADEC2HADEC;
END_VAR
TEST('Golden_Tenerife_2026');
fb(jd := 2461300.75, ra := 83.63, dec := 22.01, lon := -16.5, dut1 := 0.0);
CheckAngle(345.6575630310487, fb.ha_out, 1.0E-7, 'Tenerife_2026 ha');
CheckNear(22.02849232968123, fb.dec_out, 1.0E-7, 'Tenerife_2026 dec');
CheckSeparation(345.65746144326204, 22.028485286326138, fb.ha_out, fb.dec_out, 0.0002, 'Tenerife_2026 vs erfa');
TEST_FINISHED();
END_METHOD

METHOD PRIVATE Golden_Tenerife_low
VAR
	fb	: AstroBROT.FB_RADEC2HADEC;
END_VAR
TEST('Golden_Tenerife_low');
fb(jd := 2461300.75, ra := 130.0, dec := -10.0, lon := -16.5, dut1 := 0.0);
CheckAngle(299.37201176540054, fb.ha_out, 1.0E-7, 'Tenerife_low ha');
CheckNear(-10.091922210560911, fb.dec_out, 1.0E-7, 'Tenerife_low dec');
CheckSeparation(299.3719555337581, -10.091909866750818, fb.ha_out, fb.dec_out, 0.0002, 'Tenerife_low vs erfa');
TEST_FINISHED();
END_METHOD

METHOD PRIVATE Golden_South_2010
VAR
	fb	: AstroBROT.FB_RADEC2HADEC;
END_VAR
TEST('Golden_South_2010');
fb(jd := 2455197.5, ra := 312.5, dec := -47.3, lon := -70.7, dut1 := 0.0);
CheckAngle(77.17023586398261, fb.ha_out, 1.0E-7, 'South_2010 ha');
CheckNear(-47.26426875549772, fb.dec_out, 1.0E-7, 'South_2010 dec');
CheckSeparation(77.17019695311718, -47.26432489859199, fb.ha_out, fb.dec_out, 0.0002, 'South_2010 vs erfa');
TEST_FINISHED();
END_METHOD

METHOD PRIVATE Golden_Dut1
VAR
	fb	: AstroBROT.FB_RADEC2HADEC;
END_VAR
TEST('Golden_Dut1');
fb(jd := 2461300.75, ra := 83.63, dec := 22.01, lon := -16.5, dut1 := 0.9);
CheckAngle(345.6613233618934, fb.ha_out, 1.0E-7, 'Tenerife_dut1_plus ha');
CheckNear(22.02849232968123, fb.dec_out, 1.0E-7, 'Tenerife_dut1_plus dec');
CheckSeparation(345.66122170868215, 22.028485288193934, fb.ha_out, fb.dec_out, 0.0002, 'Tenerife_dut1_plus vs erfa');
fb(jd := 2461300.75, ra := 83.63, dec := 22.01, lon := -16.5, dut1 := -0.9);
CheckAngle(345.65380270020404, fb.ha_out, 1.0E-7, 'Tenerife_dut1_minus ha');
CheckNear(22.02849232968123, fb.dec_out, 1.0E-7, 'Tenerife_dut1_minus dec');
CheckSeparation(345.653701177839, 22.028485284458373, fb.ha_out, fb.dec_out, 0.0002, 'Tenerife_dut1_minus vs erfa');
TEST_FINISHED();
END_METHOD

METHOD PRIVATE Golden_RA_Wrap
VAR
	fb	: AstroBROT.FB_RADEC2HADEC;
END_VAR
TEST('Golden_RA_Wrap');
fb(jd := 2461300.75, ra := 0.0001, dec := 22.01, lon := -16.5, dut1 := 0.0);
CheckAngle(69.34278166497118, fb.ha_out, 1.0E-7, 'RA_wrap_low ha');
CheckNear(22.16156103752678, fb.dec_out, 1.0E-7, 'RA_wrap_low dec');
CheckSeparation(69.34272927043514, 22.16158906186533, fb.ha_out, fb.dec_out, 0.0002, 'RA_wrap_low vs erfa');
fb(jd := 2461300.75, ra := 359.9999, dec := 22.01, lon := -16.5, dut1 := 0.0);
CheckAngle(69.34298187519398, fb.ha_out, 1.0E-7, 'RA_wrap_high ha');
CheckNear(22.16156103790214, fb.dec_out, 1.0E-7, 'RA_wrap_high dec');
CheckSeparation(69.34292948093092, 22.161589062278132, fb.ha_out, fb.dec_out, 0.0002, 'RA_wrap_high vs erfa');
TEST_FINISHED();
END_METHOD

METHOD PRIVATE Golden_Poles
VAR
	fb	: AstroBROT.FB_RADEC2HADEC;
END_VAR
TEST('Golden_Poles');
fb(jd := 2461300.75, ra := 0.0, dec := 90.0, lon := -16.5, dut1 := 0.0);
CheckAngle(250.63644034864151, fb.ha_out, 1.0E-7, 'North_pole ha');
CheckNear(89.85080571177119, fb.dec_out, 1.0E-7, 'North_pole dec');
CheckSeparation(250.63721443708533, 89.8507228178902, fb.ha_out, fb.dec_out, 0.0002, 'North_pole vs erfa');
fb(jd := 2455197.5, ra := 0.0, dec := -90.0, lon := -70.7, dut1 := 0.0);
CheckAngle(29.9862312944732, fb.ha_out, 1.0E-7, 'South_pole ha');
CheckNear(-89.94820320442783, fb.dec_out, 1.0E-7, 'South_pole dec');
CheckSeparation(29.899988989677052, -89.94824504562501, fb.ha_out, fb.dec_out, 0.0002, 'South_pole vs erfa');
TEST_FINISHED();
END_METHOD

METHOD PRIVATE Golden_Near_The_Poles
VAR
	fb	: AstroBROT.FB_RADEC2HADEC;
END_VAR
TEST('Golden_Near_The_Poles');
fb(jd := 2461300.75, ra := 200.0, dec := 89.9, lon := -16.5, dut1 := 0.0);
CheckAngle(242.11458567841964, fb.ha_out, 1.0E-7, 'Near_north_pole ha');
CheckNear(89.75492331909197, fb.dec_out, 1.0E-7, 'Near_north_pole dec');
CheckSeparation(242.12047093980044, 89.75484732066303, fb.ha_out, fb.dec_out, 0.0002, 'Near_north_pole vs erfa');
fb(jd := 2455197.5, ra := 200.0, dec := -89.9, lon := -70.7, dut1 := 0.0);
CheckAngle(170.60136769350444, fb.ha_out, 1.0E-7, 'Near_south_pole ha');
CheckNear(-89.94559816252283, fb.dec_out, 1.0E-7, 'Near_south_pole dec');
CheckSeparation(170.55436891323328, -89.9455612839385, fb.ha_out, fb.dec_out, 0.0002, 'Near_south_pole vs erfa');
TEST_FINISHED();
END_METHOD

METHOD PRIVATE Right_Ascension_Is_Periodic
VAR
	fb	: AstroBROT.FB_RADEC2HADEC;
END_VAR
TEST('Right_Ascension_Is_Periodic');
// ra and ra +- 360 are the same position
fb(jd := 2461300.75, ra := -276.37, dec := 22.01, lon := -16.5);
CheckAngle(345.6575630310487, fb.ha_out, 1.0E-9, 'ra - 360 ha');
CheckNear(22.02849232968123, fb.dec_out, 1.0E-9, 'ra - 360 dec');
fb(jd := 2461300.75, ra := 443.63, dec := 22.01, lon := -16.5);
CheckAngle(345.6575630310487, fb.ha_out, 1.0E-9, 'ra + 360 ha');
CheckNear(22.02849232968123, fb.dec_out, 1.0E-9, 'ra + 360 dec');
TEST_FINISHED();
END_METHOD

METHOD PRIVATE Longitude_Is_Periodic
VAR
	fb	: AstroBROT.FB_RADEC2HADEC;
END_VAR
TEST('Longitude_Is_Periodic');
// lon and lon +- 360 are the same place
fb(jd := 2461300.75, ra := 83.63, dec := 22.01, lon := 343.5);
CheckAngle(345.6575630310487, fb.ha_out, 1.0E-9, 'lon + 360 ha');
fb(jd := 2461300.75, ra := 83.63, dec := 22.01, lon := -376.5);
CheckAngle(345.6575630310487, fb.ha_out, 1.0E-9, 'lon - 360 ha');
TEST_FINISHED();
END_METHOD

METHOD PRIVATE Outputs_Stay_In_Range
VAR
	fb	: AstroBROT.FB_RADEC2HADEC;
	i	: INT;
	fRa	: LREAL;
END_VAR
TEST('Outputs_Stay_In_Range');
// a sweep over the whole RA circle and the declinations up to and including the poles
FOR i := 0 TO 8 DO
	fRa := 45.0 * i;
	fb(jd := 2461300.75, ra := fRa, dec := 90.0, lon := -16.5);
	AssertTrue(Condition := fb.ha_out >= 0.0 AND fb.ha_out < 360.0 AND fb.dec_out <= 90.0 AND fb.dec_out >= -90.0, Message := 'ra sweep at dec +90 stays in range');
	fb(jd := 2461300.75, ra := fRa, dec := -90.0, lon := -16.5);
	AssertTrue(Condition := fb.ha_out >= 0.0 AND fb.ha_out < 360.0 AND fb.dec_out <= 90.0 AND fb.dec_out >= -90.0, Message := 'ra sweep at dec -90 stays in range');
	fb(jd := 2461300.75, ra := fRa, dec := 0.0, lon := -16.5);
	AssertTrue(Condition := fb.ha_out >= 0.0 AND fb.ha_out < 360.0 AND fb.dec_out <= 90.0 AND fb.dec_out >= -90.0, Message := 'ra sweep at dec 0 stays in range');
END_FOR
TEST_FINISHED();
END_METHOD

METHOD PRIVATE Time_Inputs_Are_Not_Modified
VAR
	fb	: AstroBROT.FB_RADEC2HADEC;
END_VAR
TEST('Time_Inputs_Are_Not_Modified');
fb(jd := 2461300.75, ra := 83.63, dec := 22.01, lon := -16.5, dut1 := 0.5);
CheckNear(2461300.75, fb.jd, 0.0, 'jd unchanged');
CheckNear(-16.5, fb.lon, 0.0, 'lon unchanged');
CheckNear(0.5, fb.dut1, 0.0, 'dut1 unchanged');
TEST_FINISHED();
END_METHOD

END_FUNCTION_BLOCK

// ---- POUs/FB_HADEC2RADEC_Tests.TcPOU
// Tests for AstroBROT.FB_HADEC2RADEC (apparent hour angle / Dec -> ICRS RA/Dec; the block IAG50cm uses).
//
// GENERATED by AstroBROT/testing/gen_block_tests.py from testing/golden_blocks.py, do not edit the numbers by hand.
// Every golden case is checked against the Python port of the ST (1E-7 deg) and against erfa.atoc13 as a great-circle
// separation on the sky (2E-4 deg = 0.72 arcsec).
//
// KNOWN LIMITATION, pinned here on purpose: at exactly dec = +-90 the ST applies the aberration and nutation
// corrections in (ra, dec), d_ra grows like 1/cos(dec) and the dec correction is evaluated at an RA that means
// nothing there. The result then depends on the hour angle and is 4.7 arcsec (north) / 39 arcsec (south) away from
// erfa. Golden_Exact_Poles allows 0.015 deg so that it cannot get worse unnoticed; 0.1 deg from the pole the error is
// back at 0.5 arcsec (Golden_Near_The_Poles, strict tolerance).
FUNCTION_BLOCK FB_HADEC2RADEC_Tests EXTENDS TcUnit.FB_TestSuite
VAR
END_VAR

